LIN {X 0,Y 192.698,Z 291.389,A -85,B 0,C 180,E1 -21893.011,E2 -21893.011} C_VEL
LIN {X 0,Y 200.351,Z 314.138,A -85,B 0,C 180,E1 -21894.699,E2 -21894.699} C_VEL
LIN {X 0,Y 198.491,Z 360.871,A -85,B 0,C 180,E1 -21896.755,E2 -21896.755} C_VEL
LIN {X 0,Y 197.875,Z 372.653,A -85,B 0,C 180,E1 -21897.641,E2 -21897.641} C_VEL
LIN {X 0,Y 196.951,Z 382.953,A -85,B 0,C 180,E1 -21898.798,E2 -21898.798} C_VEL
LIN {X 0,Y 196.113,Z 391.868,A -85,B 0,C 180,E1 -21900.112,E2 -21900.112} C_VEL
LIN {X 0,Y 195.247,Z 399.913,A -85,B 0,C 180,E1 -21901.591,E2 -21901.591} C_VEL
LIN {X 0,Y 194.171,Z 407.148,A -85,B 0,C 180,E1 -21903.2,E2 -21903.2} C_VEL
LIN {X 0,Y 193.185,Z 414.142,A -85,B 0,C 180,E1 -21905.09,E2 -21905.09} C_VEL
LIN {X 0,Y 192.435,Z 419.904,A -85,B 0,C 180,E1 -21906.965,E2 -21906.965} C_VEL
LIN {X 0,Y 191.676,Z 425.271,A -85,B 0,C 180,E1 -21909.054,E2 -21909.054} C_VEL
LIN {X 0,Y 191.095,Z 430.313,A -85,B 0,C 180,E1 -21911.451,E2 -21911.451} C_VEL
LIN {X 0,Y 190.631,Z 434.006,A -85,B 0,C 180,E1 -21913.608,E2 -21913.608} C_VEL
LIN {X 0,Y 190.248,Z 437.996,A -85,B 0,C 180,E1 -21916.63,E2 -21916.63} C_VEL
LIN {X 0,Y 190.193,Z 439.702,A -85,B 0,C 180,E1 -21918.31,E2 -21918.31} C_VEL
LIN {X 0,Y 190.411,Z 441.761,A -85,B 0,C 180,E1 -21921.14,E2 -21921.14} C_VEL
LIN {X 0,Y 190.952,Z 442.925,A -85,B 0,C 180,E1 -21924.065,E2 -21924.065} C_VEL
LIN {X 0,Y 192.023,Z 443.094,A -85,B 0,C 180,E1 -21927.327,E2 -21927.327} C_VEL
LIN {X 0,Y 193.605,Z 442.067,A -85,B 0,C 180,E1 -21930.597,E2 -21930.597} C_VEL
LIN {X 0,Y 196.19,Z 438.937,A -85,B 0,C 180,E1 -21934.543,E2 -21934.543} C_VEL
LIN {X 0,Y 198.352,Z 435.744,A -85,B 0,C 180,E1 -21937.103,E2 -21937.103} C_VEL
LIN {X 0,Y 200.792,Z 431.697,A -85,B 0,C 180,E1 -21939.514,E2 -21939.514} C_VEL
LIN {X 0,Y 204.205,Z 425.453,A -85,B 0,C 180,E1 -21942.311,E2 -21942.311} C_VEL
LIN {X 0,Y 207.631,Z 417.988,A -85,B 0,C 180,E1 -21944.791,E2 -21944.791} C_VEL
LIN {X 0,Y 210.688,Z 410.33,A -85,B 0,C 180,E1 -21946.744,E2 -21946.744} C_VEL
LIN {X 0,Y 212.919,Z 403.856,A -85,B 0,C 180,E1 -21948.096,E2 -21948.096} C_VEL
LIN {X 0,Y 215.546,Z 395.131,A -85,B 0,C 180,E1 -21949.555,E2 -21949.555} C_VEL
LIN {X 0,Y 217.706,Z 386.417,A -85,B 0,C 180,E1 -21950.713,E2 -21950.713} C_VEL
LIN {X 0,Y 219.864,Z 375.243,A -85,B 0,C 180,E1 -21951.841,E2 -21951.841} C_VEL
LIN {X 0,Y 221.31,Z 363.987,A -85,B 0,C 180,E1 -21952.591,E2 -21952.591} C_VEL
LIN {X 0,Y 223.453,Z 336.581,A -85,B 0,C 180,E1 -21953.743,E2 -21953.743} C_VEL
LIN {X 0,Y 217.6,Z 325.466,A -85,B 0,C 180,E1 -21956.298,E2 -21956.298} C_VEL
LIN {X 0,Y 214.117,Z 319.83,A -85,B 0,C 180,E1 -21957.946,E2 -21957.946} C_VEL
LIN {X 0,Y 210.484,Z 314.361,A -85,B 0,C 180,E1 -21959.803,E2 -21959.803} C_VEL
LIN {X 0,Y 208.514,Z 311.193,A -85,B 0,C 180,E1 -21960.926,E2 -21960.926} C_VEL
LIN {X 0,Y 205.81,Z 307.32,A -85,B 0,C 180,E1 -21962.525,E2 -21962.525} C_VEL
LIN {X 0,Y 203.157,Z 304.407,A -85,B 0,C 180,E1 -21964.217,E2 -21964.217} C_VEL
LIN {X 0,Y 202.125,Z 302.631,A -85,B 0,C 180,E1 -21964.988,E2 -21964.988} C_VEL
LIN {X 0,Y 199.456,Z 300.395,A -85,B 0,C 180,E1 -21966.896,E2 -21966.896} C_VEL
LIN {X 0,Y 197.961,Z 297.373,A -85,B 0,C 180,E1 -21968.339,E2 -21968.339} C_VEL
LIN {X 0,Y 194.198,Z 294.632,A -85,B 0,C 180,E1 -21971.987,E2 -21971.987} C_VEL
LIN {X 0,Y 193.008,Z 292.406,A -85,B 0,C 180,E1 -21973.693,E2 -21973.693} C_VEL
LIN {X 0,Y 192.795,Z 291.28,A -85,B 0,C 180,E1 -21974.246,E2 -21974.246} C_VEL
LIN {X 0,Y 192.71,Z 291.289,A -85,B 0,C 180,E1 -21979.163,E2 -21979.163} C_VEL
LIN {X 0,Y 192.662,Z 291.287,A -85,B 0,C 180,E1 -21984.226,E2 -21984.226} C_VEL
LIN {X 0,Y 192.64,Z 291.29,A -85,B 0,C 180,E1 -21988.889,E2 -21988.889} C_VEL
LIN {X 0,Y 193.831,Z 294.774,A -85,B 0,C 180,E1 -21995.462,E2 -21995.462} C_VEL
LIN {X 0,Y 194.221,Z 295.838,A -85,B 0,C 180,E1 -21996.347,E2 -21996.347} C_VEL
LIN {X 0,Y 199.63,Z 303.251,A -85,B 0,C 180,E1 -22001.645,E2 -22001.645} C_VEL
LIN {X 0,Y 203.657,Z 309.45,A -85,B 0,C 180,E1 -22004.662,E2 -22004.662} C_VEL
LIN {X 0,Y 208.105,Z 316.783,A -85,B 0,C 180,E1 -22007.468,E2 -22007.468} C_VEL
LIN {X 0,Y 211.698,Z 323.218,A -85,B 0,C 180,E1 -22009.493,E2 -22009.493} C_VEL
LIN {X 0,Y 215.585,Z 330.908,A -85,B 0,C 180,E1 -22011.482,E2 -22011.482} C_VEL
LIN {X 0,Y 220.085,Z 341.471,A -85,B 0,C 180,E1 -22013.657,E2 -22013.657} C_VEL
LIN {X 0,Y 221.449,Z 354.874,A -85,B 0,C 180,E1 -22014.901,E2 -22014.901} C_VEL
LIN {X 0,Y 221.826,Z 363.402,A -85,B 0,C 180,E1 -22015.531,E2 -22015.531} C_VEL
LIN {X 0,Y 221.197,Z 371.063,A -85,B 0,C 180,E1 -22015.822,E2 -22015.822} C_VEL
LIN {X 0,Y 220.14,Z 376.884,A -85,B 0,C 180,E1 -22015.915,E2 -22015.915} C_VEL
LIN {X 0,Y 216.946,Z 386.292,A -85,B 0,C 180,E1 -22015.875,E2 -22015.875} C_VEL
LIN {X 0,Y 213.279,Z 395.447,A -85,B 0,C 180,E1 -22016.008,E2 -22016.008} C_VEL
LIN {X 0,Y 211.5,Z 400.855,A -85,B 0,C 180,E1 -22016.403,E2 -22016.403} C_VEL
LIN {X 0,Y 208.494,Z 411.167,A -85,B 0,C 180,E1 -22017.649,E2 -22017.649} C_VEL
LIN {X 0,Y 205.745,Z 419.123,A -85,B 0,C 180,E1 -22018.893,E2 -22018.893} C_VEL
LIN {X 0,Y 202.813,Z 426.763,A -85,B 0,C 180,E1 -22020.411,E2 -22020.411} C_VEL
LIN {X 0,Y 198.982,Z 435.728,A -85,B 0,C 180,E1 -22022.668,E2 -22022.668} C_VEL
LIN {X 0,Y 195.446,Z 442.776,A -85,B 0,C 180,E1 -22025.008,E2 -22025.008} C_VEL
LIN {X 0,Y 192.345,Z 448.444,A -85,B 0,C 180,E1 -22027.441,E2 -22027.441} C_VEL
LIN {X 0,Y 189.195,Z 453.782,A -85,B 0,C 180,E1 -22030.47,E2 -22030.47} C_VEL
LIN {X 0,Y 186.736,Z 457.778,A -85,B 0,C 180,E1 -22033.605,E2 -22033.605} C_VEL
LIN {X 0,Y 184.977,Z 460.546,A -85,B 0,C 180,E1 -22036.824,E2 -22036.824} C_VEL
LIN {X 0,Y 184.163,Z 461.689,A -85,B 0,C 180,E1 -22039.001,E2 -22039.001} C_VEL
LIN {X 0,Y 183.645,Z 462.356,A -85,B 0,C 180,E1 -22041.195,E2 -22041.195} C_VEL
LIN {X 0,Y 183.328,Z 462.409,A -85,B 0,C 180,E1 -22045.381,E2 -22045.381} C_VEL
LIN {X 0,Y 183.47,Z 461.54,A -85,B 0,C 180,E1 -22047.805,E2 -22047.805} C_VEL
LIN {X 0,Y 183.571,Z 460.179,A -85,B 0,C 180,E1 -22050.001,E2 -22050.001} C_VEL
LIN {X 0,Y 183.601,Z 457.145,A -85,B 0,C 180,E1 -22053.292,E2 -22053.292} C_VEL
LIN {X 0,Y 183.609,Z 452.606,A -85,B 0,C 180,E1 -22056.594,E2 -22056.594} C_VEL
LIN {X 0,Y 183.92,Z 447.511,A -85,B 0,C 180,E1 -22059.347,E2 -22059.347} C_VEL
LIN {X 0,Y 184.381,Z 442.506,A -85,B 0,C 180,E1 -22061.544,E2 -22061.544} C_VEL
LIN {X 0,Y 185.122,Z 436.463,A -85,B 0,C 180,E1 -22063.726,E2 -22063.726} C_VEL
LIN {X 0,Y 186.263,Z 428.077,A -85,B 0,C 180,E1 -22066.157,E2 -22066.157} C_VEL
LIN {X 0,Y 187.402,Z 420.033,A -85,B 0,C 180,E1 -22068.023,E2 -22068.023} C_VEL
LIN {X 0,Y 188.624,Z 409.933,A -85,B 0,C 180,E1 -22069.876,E2 -22069.876} C_VEL
LIN {X 0,Y 189.99,Z 399.38,A -85,B 0,C 180,E1 -22071.283,E2 -22071.283} C_VEL
LIN {X 0,Y 190.803,Z 389.702,A -85,B 0,C 180,E1 -22072.245,E2 -22072.245} C_VEL
LIN {X 0,Y 191.446,Z 379.539,A -85,B 0,C 180,E1 -22072.939,E2 -22072.939} C_VEL
LIN {X 0,Y 192.199,Z 354.528,A -85,B 0,C 180,E1 -22074.102,E2 -22074.102} C_VEL
LIN {X 0,Y 187.917,Z 303.799,A -85,B 0,C 180,E1 -22076.892,E2 -22076.892} C_VEL
LIN {X 0,Y 186.171,Z 294.826,A -85,B 0,C 180,E1 -22081.396,E2 -22081.396} C_VEL
LIN {X 0,Y 185.691,Z 292.169,A -85,B 0,C 180,E1 -22082.815,E2 -22082.815} C_VEL
LIN {X 0,Y 185.548,Z 292.184,A -85,B 0,C 180,E1 -22087.303,E2 -22087.303} C_VEL
LIN {X 0,Y 185.488,Z 292.19,A -85,B 0,C 180,E1 -22090.729,E2 -22090.729} C_VEL
LIN {X 0,Y 185.462,Z 292.195,A -85,B 0,C 180,E1 -22096.054,E2 -22096.054} C_VEL
LIN {X 0,Y 185.469,Z 292.192,A -85,B 0,C 180,E1 -22099.894,E2 -22099.894} C_VEL
LIN {X 0,Y 185.508,Z 292.186,A -85,B 0,C 180,E1 -22102.71,E2 -22102.71} C_VEL
LIN {X 0,Y 185.545,Z 292.183,A -85,B 0,C 180,E1 -22107.973,E2 -22107.973} C_VEL
LIN {X 0,Y 185.583,Z 292.175,A -85,B 0,C 180,E1 -22110.575,E2 -22110.575} C_VEL
LIN {X 0,Y 185.589,Z 292.18,A -85,B 0,C 180,E1 -22115.381,E2 -22115.381} C_VEL
LIN {X 0,Y 185.675,Z 292.167,A -85,B 0,C 180,E1 -22121.132,E2 -22121.132} C_VEL
LIN {X 0,Y 185.694,Z 292.164,A -85,B 0,C 180,E1 -22124.635,E2 -22124.635} C_VEL
LIN {X 0,Y 185.888,Z 292.141,A -85,B 0,C 180,E1 -22129.416,E2 -22129.416} C_VEL
LIN {X 0,Y 185.947,Z 292.135,A -85,B 0,C 180,E1 -22133.488,E2 -22133.488} C_VEL
LIN {X 0,Y 186.205,Z 292.103,A -85,B 0,C 180,E1 -22137.835,E2 -22137.835} C_VEL
LIN {X 0,Y 186.405,Z 292.078,A -85,B 0,C 180,E1 -22139.998,E2 -22139.998} C_VEL
LIN {X 0,Y 185.923,Z 292.134,A -85,B 0,C 180,E1 -22144.334,E2 -22144.334} C_VEL
LIN {X 0,Y 186.011,Z 292.125,A -85,B 0,C 180,E1 -22148.691,E2 -22148.691} C_VEL
LIN {X 0,Y 185.731,Z 292.157,A -85,B 0,C 180,E1 -22153.121,E2 -22153.121} C_VEL
LIN {X 0,Y 185.707,Z 292.162,A -85,B 0,C 180,E1 -22158.897,E2 -22158.897} C_VEL
LIN {X 0,Y 185.597,Z 292.177,A -85,B 0,C 180,E1 -22164.66,E2 -22164.66} C_VEL
LIN {X 0,Y 185.575,Z 292.178,A -85,B 0,C 180,E1 -22169.491,E2 -22169.491} C_VEL
LIN {X 0,Y 185.516,Z 292.187,A -85,B 0,C 180,E1 -22174.626,E2 -22174.626} C_VEL
LIN {X 0,Y 185.539,Z 292.183,A -85,B 0,C 180,E1 -22177.302,E2 -22177.302} C_VEL
LIN {X 0,Y 185.524,Z 292.186,A -85,B 0,C 180,E1 -22180.744,E2 -22180.744} C_VEL
LIN {X 0,Y 185.559,Z 292.179,A -85,B 0,C 180,E1 -22186.02,E2 -22186.02} C_VEL
LIN {X 0,Y 185.536,Z 292.187,A -85,B 0,C 180,E1 -22189.913,E2 -22189.913} C_VEL
LIN {X 0,Y 185.554,Z 292.181,A -85,B 0,C 180,E1 -22192.699,E2 -22192.699} C_VEL
LIN {X 0,Y 185.539,Z 292.186,A -85,B 0,C 180,E1 -22197.974,E2 -22197.974} C_VEL
LIN {X 0,Y 185.576,Z 292.179,A -85,B 0,C 180,E1 -22200.575,E2 -22200.575} C_VEL
LIN {X 0,Y 185.581,Z 292.178,A -85,B 0,C 180,E1 -22205.382,E2 -22205.382} C_VEL
LIN {X 0,Y 185.669,Z 292.166,A -85,B 0,C 180,E1 -22211.132,E2 -22211.132} C_VEL
LIN {X 0,Y 185.718,Z 292.162,A -85,B 0,C 180,E1 -22214.639,E2 -22214.639} C_VEL
LIN {X 0,Y 185.918,Z 292.136,A -85,B 0,C 180,E1 -22219.358,E2 -22219.358} C_VEL
LIN {X 0,Y 185.954,Z 292.134,A -85,B 0,C 180,E1 -22223.489,E2 -22223.489} C_VEL
LIN {X 0,Y 186.2,Z 292.1,A -85,B 0,C 180,E1 -22227.836,E2 -22227.836} C_VEL
LIN {X 0,Y 186.4,Z 292.077,A -85,B 0,C 180,E1 -22229.999,E2 -22229.999} C_VEL
LIN {X 0,Y 185.916,Z 292.137,A -85,B 0,C 180,E1 -22234.335,E2 -22234.335} C_VEL
LIN {X 0,Y 186.001,Z 292.125,A -85,B 0,C 180,E1 -22238.692,E2 -22238.692} C_VEL
LIN {X 0,Y 185.757,Z 292.157,A -85,B 0,C 180,E1 -22243.12,E2 -22243.12} C_VEL
LIN {X 0,Y 185.682,Z 292.169,A -85,B 0,C 180,E1 -22247.625,E2 -22247.625} C_VEL
LIN {X 0,Y 185.609,Z 292.177,A -85,B 0,C 180,E1 -22252.395,E2 -22252.395} C_VEL
LIN {X 0,Y 193.402,Z 315.234,A -85,B 0,C 180,E1 -22254.206,E2 -22254.206} C_VEL
LIN {X 0,Y 191.595,Z 360.842,A -85,B 0,C 180,E1 -22256.287,E2 -22256.287} C_VEL
LIN {X 0,Y 190.952,Z 372.604,A -85,B 0,C 180,E1 -22257.185,E2 -22257.185} C_VEL
LIN {X 0,Y 189.931,Z 383.741,A -85,B 0,C 180,E1 -22258.481,E2 -22258.481} C_VEL
LIN {X 0,Y 189.094,Z 392.381,A -85,B 0,C 180,E1 -22259.807,E2 -22259.807} C_VEL
LIN {X 0,Y 188.286,Z 399.565,A -85,B 0,C 180,E1 -22261.159,E2 -22261.159} C_VEL
LIN {X 0,Y 187.086,Z 407.606,A -85,B 0,C 180,E1 -22263.003,E2 -22263.003} C_VEL
LIN {X 0,Y 186.151,Z 414.112,A -85,B 0,C 180,E1 -22264.821,E2 -22264.821} C_VEL
LIN {X 0,Y 185.456,Z 419.331,A -85,B 0,C 180,E1 -22266.543,E2 -22266.543} C_VEL
LIN {X 0,Y 184.608,Z 425.155,A -85,B 0,C 180,E1 -22268.847,E2 -22268.847} C_VEL
LIN {X 0,Y 184.064,Z 429.983,A -85,B 0,C 180,E1 -22271.172,E2 -22271.172} C_VEL
LIN {X 0,Y 183.527,Z 434.046,A -85,B 0,C 180,E1 -22273.572,E2 -22273.572} C_VEL
LIN {X 0,Y 183.192,Z 437.698,A -85,B 0,C 180,E1 -22276.329,E2 -22276.329} C_VEL
LIN {X 0,Y 183.143,Z 440.57,A -85,B 0,C 180,E1 -22279.283,E2 -22279.283} C_VEL
LIN {X 0,Y 183.707,Z 443.063,A -85,B 0,C 180,E1 -22283.453,E2 -22283.453} C_VEL
LIN {X 0,Y 184.706,Z 443.638,A -85,B 0,C 180,E1 -22286.831,E2 -22286.831} C_VEL
LIN {X 0,Y 186.495,Z 442.813,A -85,B 0,C 180,E1 -22290.668,E2 -22290.668} C_VEL
LIN {X 0,Y 189.185,Z 440.155,A -85,B 0,C 180,E1 -22294.81,E2 -22294.81} C_VEL
LIN {X 0,Y 191.728,Z 436.783,A -85,B 0,C 180,E1 -22297.764,E2 -22297.764} C_VEL
LIN {X 0,Y 194.21,Z 432.995,A -85,B 0,C 180,E1 -22300.195,E2 -22300.195} C_VEL
LIN {X 0,Y 196.798,Z 428.706,A -85,B 0,C 180,E1 -22302.323,E2 -22302.323} C_VEL
LIN {X 0,Y 200.044,Z 422.512,A -85,B 0,C 180,E1 -22304.725,E2 -22304.725} C_VEL
LIN {X 0,Y 202.863,Z 416.534,A -85,B 0,C 180,E1 -22306.569,E2 -22306.569} C_VEL
LIN {X 0,Y 206.102,Z 408.688,A -85,B 0,C 180,E1 -22308.51,E2 -22308.51} C_VEL
LIN {X 0,Y 209.448,Z 399.12,A -85,B 0,C 180,E1 -22310.343,E2 -22310.343} C_VEL
LIN {X 0,Y 212.119,Z 389.409,A -85,B 0,C 180,E1 -22311.746,E2 -22311.746} C_VEL
LIN {X 0,Y 214.281,Z 379.683,A -85,B 0,C 180,E1 -22312.809,E2 -22312.809} C_VEL
LIN {X 0,Y 215.719,Z 370.797,A -85,B 0,C 180,E1 -22313.557,E2 -22313.557} C_VEL
LIN {X 0,Y 217.003,Z 359.592,A -85,B 0,C 180,E1 -22314.202,E2 -22314.202} C_VEL
LIN {X 0,Y 218.549,Z 339.503,A -85,B 0,C 180,E1 -22315.032,E2 -22315.032} C_VEL
LIN {X 0,Y 213.644,Z 329.87,A -85,B 0,C 180,E1 -22317.38,E2 -22317.38} C_VEL
LIN {X 0,Y 210.475,Z 324.818,A -85,B 0,C 180,E1 -22318.96,E2 -22318.96} C_VEL
LIN {X 0,Y 205.715,Z 317.082,A -85,B 0,C 180,E1 -22321.704,E2 -22321.704} C_VEL
LIN {X 0,Y 203.329,Z 313.604,A -85,B 0,C 180,E1 -22323.211,E2 -22323.211} C_VEL
LIN {X 0,Y 200.543,Z 310.193,A -85,B 0,C 180,E1 -22325.122,E2 -22325.122} C_VEL
LIN {X 0,Y 199.619,Z 308.946,A -85,B 0,C 180,E1 -22325.811,E2 -22325.811} C_VEL
LIN {X 0,Y 196.979,Z 306.174,A -85,B 0,C 180,E1 -22327.932,E2 -22327.932} C_VEL
LIN {X 0,Y 195.858,Z 303.828,A -85,B 0,C 180,E1 -22329.095,E2 -22329.095} C_VEL
LIN {X 0,Y 192.674,Z 301.456,A -85,B 0,C 180,E1 -22332.365,E2 -22332.365} C_VEL
LIN {X 0,Y 191.317,Z 298.86,A -85,B 0,C 180,E1 -22334.426,E2 -22334.426} C_VEL
LIN {X 0,Y 191.071,Z 298.182,A -85,B 0,C 180,E1 -22334.922,E2 -22334.922} C_VEL
LIN {X 0,Y 188.225,Z 296.835,A -85,B 0,C 180,E1 -22341.926,E2 -22341.926} C_VEL
LIN {X 0,Y 188.284,Z 296.943,A -85,B 0,C 180,E1 -22346.612,E2 -22346.612} C_VEL
LIN {X 0,Y 188.963,Z 297.537,A -85,B 0,C 180,E1 -22349.221,E2 -22349.221} C_VEL
LIN {X 0,Y 192.232,Z 301.815,A -85,B 0,C 180,E1 -22355.319,E2 -22355.319} C_VEL
LIN {X 0,Y 197.076,Z 308.988,A -85,B 0,C 180,E1 -22360.605,E2 -22360.605} C_VEL
LIN {X 0,Y 201.683,Z 316.494,A -85,B 0,C 180,E1 -22364.286,E2 -22364.286} C_VEL
LIN {X 0,Y 205.401,Z 322.922,A -85,B 0,C 180,E1 -22366.76,E2 -22366.76} C_VEL
LIN {X 0,Y 208.337,Z 328.367,A -85,B 0,C 180,E1 -22368.53,E2 -22368.53} C_VEL
LIN {X 0,Y 212.02,Z 336.084,A -85,B 0,C 180,E1 -22370.57,E2 -22370.57} C_VEL
LIN {X 0,Y 215.656,Z 345.058,A -85,B 0,C 180,E1 -22372.499,E2 -22372.499} C_VEL
LIN {X 0,Y 216.746,Z 357.398,A -85,B 0,C 180,E1 -22373.663,E2 -22373.663} C_VEL
LIN {X 0,Y 216.993,Z 364.53,A -85,B 0,C 180,E1 -22374.197,E2 -22374.197} C_VEL
LIN {X 0,Y 215.208,Z 382.567,A -85,B 0,C 180,E1 -22374.972,E2 -22374.972} C_VEL
LIN {X 0,Y 213.235,Z 393.234,A -85,B 0,C 180,E1 -22375.697,E2 -22375.697} C_VEL
LIN {X 0,Y 211.5,Z 400.855,A -85,B 0,C 180,E1 -22376.403,E2 -22376.403} C_VEL
LIN {X 0,Y 209.976,Z 404.484,A -85,B 0,C 180,E1 -22376.651,E2 -22376.651} C_VEL
LIN {X 0,Y 206.162,Z 410.158,A -85,B 0,C 180,E1 -22376.796,E2 -22376.796} C_VEL
LIN {X 0,Y 202.253,Z 415.631,A -85,B 0,C 180,E1 -22377.027,E2 -22377.027} C_VEL
LIN {X 0,Y 200.604,Z 418.76,A -85,B 0,C 180,E1 -22377.456,E2 -22377.456} C_VEL
LIN {X 0,Y 197.188,Z 427.239,A -85,B 0,C 180,E1 -22379.181,E2 -22379.181} C_VEL
LIN {X 0,Y 192.766,Z 436.673,A -85,B 0,C 180,E1 -22381.709,E2 -22381.709} C_VEL
LIN {X 0,Y 189.083,Z 443.41,A -85,B 0,C 180,E1 -22384.105,E2 -22384.105} C_VEL
LIN {X 0,Y 185.84,Z 448.869,A -85,B 0,C 180,E1 -22386.605,E2 -22386.605} C_VEL
LIN {X 0,Y 183.563,Z 452.459,A -85,B 0,C 180,E1 -22388.672,E2 -22388.672} C_VEL
LIN {X 0,Y 180.691,Z 456.661,A -85,B 0,C 180,E1 -22391.872,E2 -22391.872} C_VEL
LIN {X 0,Y 179.219,Z 458.757,A -85,B 0,C 180,E1 -22394.069,E2 -22394.069} C_VEL
LIN {X 0,Y 178.055,Z 460.375,A -85,B 0,C 180,E1 -22396.302,E2 -22396.302} C_VEL
LIN {X 0,Y 177.189,Z 461.48,A -85,B 0,C 180,E1 -22398.562,E2 -22398.562} C_VEL
LIN {X 0,Y 176.613,Z 462.017,A -85,B 0,C 180,E1 -22400.842,E2 -22400.842} C_VEL
LIN {X 0,Y 176.31,Z 462.112,A -85,B 0,C 180,E1 -22403.133,E2 -22403.133} C_VEL
LIN {X 0,Y 176.265,Z 461.764,A -85,B 0,C 180,E1 -22405.427,E2 -22405.427} C_VEL
LIN {X 0,Y 176.403,Z 460.922,A -85,B 0,C 180,E1 -22407.717,E2 -22407.717} C_VEL
LIN {X 0,Y 176.48,Z 458.525,A -85,B 0,C 180,E1 -22411.141,E2 -22411.141} C_VEL
LIN {X 0,Y 176.544,Z 456.246,A -85,B 0,C 180,E1 -22413.424,E2 -22413.424} C_VEL
LIN {X 0,Y 176.587,Z 451.438,A -85,B 0,C 180,E1 -22416.858,E2 -22416.858} C_VEL
LIN {X 0,Y 176.926,Z 446.182,A -85,B 0,C 180,E1 -22419.72,E2 -22419.72} C_VEL
LIN {X 0,Y 177.435,Z 440.999,A -85,B 0,C 180,E1 -22422.002,E2 -22422.002} C_VEL
LIN {X 0,Y 178.222,Z 434.749,A -85,B 0,C 180,E1 -22424.268,E2 -22424.268} C_VEL
LIN {X 0,Y 179.301,Z 427.158,A -85,B 0,C 180,E1 -22426.51,E2 -22426.51} C_VEL
LIN {X 0,Y 180.671,Z 417.781,A -85,B 0,C 180,E1 -22428.719,E2 -22428.719} C_VEL
LIN {X 0,Y 181.754,Z 408.679,A -85,B 0,C 180,E1 -22430.366,E2 -22430.366} C_VEL
LIN {X 0,Y 183.03,Z 399.064,A -85,B 0,C 180,E1 -22431.69,E2 -22431.69} C_VEL
LIN {X 0,Y 183.892,Z 389.191,A -85,B 0,C 180,E1 -22432.706,E2 -22432.706} C_VEL
LIN {X 0,Y 184.511,Z 379.499,A -85,B 0,C 180,E1 -22433.395,E2 -22433.395} C_VEL
LIN {X 0,Y 185.33,Z 355.521,A -85,B 0,C 180,E1 -22434.555,E2 -22434.555} C_VEL
LIN {X 0,Y 181.15,Z 305.379,A -85,B 0,C 180,E1 -22437.414,E2 -22437.414} C_VEL
LIN {X 0,Y 180.607,Z 303.059,A -85,B 0,C 180,E1 -22437.623,E2 -22437.623} C_VEL
LIN {X 0,Y 178.625,Z 293.049,A -85,B 0,C 180,E1 -22443.087,E2 -22443.087} C_VEL
LIN {X 0,Y 178.422,Z 293.072,A -85,B 0,C 180,E1 -22449.067,E2 -22449.067} C_VEL
LIN {X 0,Y 178.406,Z 293.07,A -85,B 0,C 180,E1 -22452.042,E2 -22452.042} C_VEL
LIN {X 0,Y 178.396,Z 293.073,A -85,B 0,C 180,E1 -22455.163,E2 -22455.163} C_VEL
LIN {X 0,Y 178.405,Z 293.073,A -85,B 0,C 180,E1 -22458.458,E2 -22458.458} C_VEL
LIN {X 0,Y 178.424,Z 293.073,A -85,B 0,C 180,E1 -22463.781,E2 -22463.781} C_VEL
LIN {X 0,Y 178.487,Z 293.063,A -85,B 0,C 180,E1 -22466.545,E2 -22466.545} C_VEL
LIN {X 0,Y 178.524,Z 293.056,A -85,B 0,C 180,E1 -22470.005,E2 -22470.005} C_VEL
LIN {X 0,Y 178.536,Z 293.057,A -85,B 0,C 180,E1 -22474.874,E2 -22474.874} C_VEL
LIN {X 0,Y 178.624,Z 293.045,A -85,B 0,C 180,E1 -22480.782,E2 -22480.782} C_VEL
LIN {X 0,Y 178.657,Z 293.037,A -85,B 0,C 180,E1 -22486.346,E2 -22486.346} C_VEL
LIN {X 0,Y 178.911,Z 293.01,A -85,B 0,C 180,E1 -22490.958,E2 -22490.958} C_VEL
LIN {X 0,Y 179.151,Z 292.982,A -85,B 0,C 180,E1 -22497.75,E2 -22497.75} C_VEL
LIN {X 0,Y 179.368,Z 292.954,A -85,B 0,C 180,E1 -22499.998,E2 -22499.998} C_VEL
LIN {X 0,Y 178.871,Z 293.012,A -85,B 0,C 180,E1 -22504.505,E2 -22504.505} C_VEL
LIN {X 0,Y 178.961,Z 293.004,A -85,B 0,C 180,E1 -22509.036,E2 -22509.036} C_VEL
LIN {X 0,Y 178.659,Z 293.04,A -85,B 0,C 180,E1 -22513.65,E2 -22513.65} C_VEL
LIN {X 0,Y 178.65,Z 293.042,A -85,B 0,C 180,E1 -22519.242,E2 -22519.242} C_VEL
LIN {X 0,Y 178.531,Z 293.058,A -85,B 0,C 180,E1 -22525.123,E2 -22525.123} C_VEL
LIN {X 0,Y 178.475,Z 293.062,A -85,B 0,C 180,E1 -22530.789,E2 -22530.789} C_VEL
LIN {X 0,Y 178.492,Z 293.063,A -85,B 0,C 180,E1 -22534.223,E2 -22534.223} C_VEL
LIN {X 0,Y 178.439,Z 293.066,A -85,B 0,C 180,E1 -22539.06,E2 -22539.06} C_VEL
LIN {X 0,Y 178.482,Z 293.065,A -85,B 0,C 180,E1 -22542.018,E2 -22542.018} C_VEL
LIN {X 0,Y 178.512,Z 293.058,A -85,B 0,C 180,E1 -22545.123,E2 -22545.123} C_VEL
LIN {X 0,Y 178.497,Z 293.061,A -85,B 0,C 180,E1 -22548.422,E2 -22548.422} C_VEL
LIN {X 0,Y 178.453,Z 293.065,A -85,B 0,C 180,E1 -22553.79,E2 -22553.79} C_VEL
LIN {X 0,Y 178.486,Z 293.062,A -85,B 0,C 180,E1 -22556.547,E2 -22556.547} C_VEL
LIN {X 0,Y 178.517,Z 293.06,A -85,B 0,C 180,E1 -22560.005,E2 -22560.005} C_VEL
LIN {X 0,Y 178.529,Z 293.056,A -85,B 0,C 180,E1 -22564.875,E2 -22564.875} C_VEL
LIN {X 0,Y 178.617,Z 293.044,A -85,B 0,C 180,E1 -22570.783,E2 -22570.783} C_VEL
LIN {X 0,Y 178.659,Z 293.043,A -85,B 0,C 180,E1 -22574.016,E2 -22574.016} C_VEL
LIN {X 0,Y 178.855,Z 293.015,A -85,B 0,C 180,E1 -22579.209,E2 -22579.209} C_VEL
LIN {X 0,Y 178.918,Z 293.009,A -85,B 0,C 180,E1 -22583.232,E2 -22583.232} C_VEL
LIN {X 0,Y 179.146,Z 292.979,A -85,B 0,C 180,E1 -22587.751,E2 -22587.751} C_VEL
LIN {X 0,Y 179.363,Z 292.954,A -85,B 0,C 180,E1 -22589.999,E2 -22589.999} C_VEL
LIN {X 0,Y 178.864,Z 293.015,A -85,B 0,C 180,E1 -22594.507,E2 -22594.507} C_VEL
LIN {X 0,Y 178.952,Z 293.003,A -85,B 0,C 180,E1 -22599.037,E2 -22599.037} C_VEL
LIN {X 0,Y 178.68,Z 293.04,A -85,B 0,C 180,E1 -22603.65,E2 -22603.65} C_VEL
LIN {X 0,Y 178.635,Z 293.044,A -85,B 0,C 180,E1 -22608.344,E2 -22608.344} C_VEL
LIN {X 0,Y 178.549,Z 293.057,A -85,B 0,C 180,E1 -22611.806,E2 -22611.806} C_VEL
LIN {X 0,Y 186.632,Z 316.9,A -85,B 0,C 180,E1 -22613.73,E2 -22613.73} C_VEL
LIN {X 0,Y 184.655,Z 361.399,A -85,B 0,C 180,E1 -22615.841,E2 -22615.841} C_VEL
LIN {X 0,Y 184.076,Z 371.745,A -85,B 0,C 180,E1 -22616.653,E2 -22616.653} C_VEL
LIN {X 0,Y 182.96,Z 384.023,A -85,B 0,C 180,E1 -22618.098,E2 -22618.098} C_VEL
LIN {X 0,Y 182.011,Z 393.352,A -85,B 0,C 180,E1 -22619.598,E2 -22619.598} C_VEL
LIN {X 0,Y 180.947,Z 401.791,A -85,B 0,C 180,E1 -22621.302,E2 -22621.302} C_VEL
LIN {X 0,Y 179.598,Z 410.629,A -85,B 0,C 180,E1 -22623.516,E2 -22623.516} C_VEL
LIN {X 0,Y 178.438,Z 418.999,A -85,B 0,C 180,E1 -22626.212,E2 -22626.212} C_VEL
LIN {X 0,Y 177.612,Z 424.689,A -85,B 0,C 180,E1 -22628.484,E2 -22628.484} C_VEL
LIN {X 0,Y 176.999,Z 429.902,A -85,B 0,C 180,E1 -22631.029,E2 -22631.029} C_VEL
LIN {X 0,Y 176.333,Z 434.957,A -85,B 0,C 180,E1 -22634.162,E2 -22634.162} C_VEL
LIN {X 0,Y 176.024,Z 438.74,A -85,B 0,C 180,E1 -22637.257,E2 -22637.257} C_VEL
LIN {X 0,Y 176.119,Z 441.438,A -85,B 0,C 180,E1 -22640.325,E2 -22640.325} C_VEL
LIN {X 0,Y 176.575,Z 443.148,A -85,B 0,C 180,E1 -22643.346,E2 -22643.346} C_VEL
LIN {X 0,Y 177.404,Z 443.964,A -85,B 0,C 180,E1 -22646.318,E2 -22646.318} C_VEL
LIN {X 0,Y 178.853,Z 443.87,A -85,B 0,C 180,E1 -22649.821,E2 -22649.821} C_VEL
LIN {X 0,Y 180.915,Z 442.453,A -85,B 0,C 180,E1 -22653.31,E2 -22653.31} C_VEL
LIN {X 0,Y 183.548,Z 439.68,A -85,B 0,C 180,E1 -22656.769,E2 -22656.769} C_VEL
LIN {X 0,Y 186.852,Z 435.408,A -85,B 0,C 180,E1 -22660.216,E2 -22660.216} C_VEL
LIN {X 0,Y 190.704,Z 429.671,A -85,B 0,C 180,E1 -22663.365,E2 -22663.365} C_VEL
LIN {X 0,Y 194.391,Z 423.134,A -85,B 0,C 180,E1 -22665.995,E2 -22665.995} C_VEL
LIN {X 0,Y 197.03,Z 417.963,A -85,B 0,C 180,E1 -22667.644,E2 -22667.644} C_VEL
LIN {X 0,Y 200.148,Z 410.948,A -85,B 0,C 180,E1 -22669.471,E2 -22669.471} C_VEL
LIN {X 0,Y 202.993,Z 403.495,A -85,B 0,C 180,E1 -22671.039,E2 -22671.039} C_VEL
LIN {X 0,Y 206.209,Z 393.646,A -85,B 0,C 180,E1 -22672.659,E2 -22672.659} C_VEL
LIN {X 0,Y 208.993,Z 382.773,A -85,B 0,C 180,E1 -22673.97,E2 -22673.97} C_VEL
LIN {X 0,Y 210.766,Z 373.08,A -85,B 0,C 180,E1 -22674.857,E2 -22674.857} C_VEL
LIN {X 0,Y 212.092,Z 363.276,A -85,B 0,C 180,E1 -22675.474,E2 -22675.474} C_VEL
LIN {X 0,Y 213.947,Z 342.669,A -85,B 0,C 180,E1 -22676.351,E2 -22676.351} C_VEL
LIN {X 0,Y 209.183,Z 333.308,A -85,B 0,C 180,E1 -22678.809,E2 -22678.809} C_VEL
LIN {X 0,Y 202.947,Z 323.019,A -85,B 0,C 180,E1 -22682.497,E2 -22682.497} C_VEL
LIN {X 0,Y 200.754,Z 319.7,A -85,B 0,C 180,E1 -22684.017,E2 -22684.017} C_VEL
LIN {X 0,Y 198.045,Z 316.092,A -85,B 0,C 180,E1 -22685.998,E2 -22685.998} C_VEL
LIN {X 0,Y 194.748,Z 312.196,A -85,B 0,C 180,E1 -22688.83,E2 -22688.83} C_VEL
LIN {X 0,Y 193.81,Z 310.422,A -85,B 0,C 180,E1 -22689.83,E2 -22689.83} C_VEL
LIN {X 0,Y 190.859,Z 307.86,A -85,B 0,C 180,E1 -22693.172,E2 -22693.172} C_VEL
LIN {X 0,Y 189.557,Z 305.072,A -85,B 0,C 180,E1 -22695.433,E2 -22695.433} C_VEL
LIN {X 0,Y 187.058,Z 303.807,A -85,B 0,C 180,E1 -22702.07,E2 -22702.07} C_VEL
LIN {X 0,Y 187.168,Z 303.955,A -85,B 0,C 180,E1 -22706.783,E2 -22706.783} C_VEL
LIN {X 0,Y 187.755,Z 304.576,A -85,B 0,C 180,E1 -22709.12,E2 -22709.12} C_VEL
LIN {X 0,Y 190.665,Z 308.622,A -85,B 0,C 180,E1 -22714.845,E2 -22714.845} C_VEL
LIN {X 0,Y 195.398,Z 316.095,A -85,B 0,C 180,E1 -22720.283,E2 -22720.283} C_VEL
LIN {X 0,Y 199.261,Z 322.715,A -85,B 0,C 180,E1 -22723.544,E2 -22723.544} C_VEL
LIN {X 0,Y 202.506,Z 328.64,A -85,B 0,C 180,E1 -22725.886,E2 -22725.886} C_VEL
LIN {X 0,Y 205.513,Z 334.477,A -85,B 0,C 180,E1 -22727.807,E2 -22727.807} C_VEL
LIN {X 0,Y 209.544,Z 343.651,A -85,B 0,C 180,E1 -22730.206,E2 -22730.206} C_VEL
LIN {X 0,Y 211.472,Z 348.859,A -85,B 0,C 180,E1 -22731.304,E2 -22731.304} C_VEL
LIN {X 0,Y 212.37,Z 363.132,A -85,B 0,C 180,E1 -22732.639,E2 -22732.639} C_VEL
LIN {X 0,Y 211.883,Z 370.305,A -85,B 0,C 180,E1 -22732.975,E2 -22732.975} C_VEL
LIN {X 0,Y 210.116,Z 384.489,A -85,B 0,C 180,E1 -22733.663,E2 -22733.663} C_VEL
LIN {X 0,Y 208.198,Z 394.072,A -85,B 0,C 180,E1 -22734.354,E2 -22734.354} C_VEL
LIN {X 0,Y 206.132,Z 402.404,A -85,B 0,C 180,E1 -22735.176,E2 -22735.176} C_VEL
LIN {X 0,Y 203.583,Z 410.576,A -85,B 0,C 180,E1 -22736.176,E2 -22736.176} C_VEL
LIN {X 0,Y 200.604,Z 418.76,A -85,B 0,C 180,E1 -22737.456,E2 -22737.456} C_VEL
LIN {X 0,Y 198.345,Z 423.523,A -85,B 0,C 180,E1 -22738.252,E2 -22738.252} C_VEL
LIN {X 0,Y 192.936,Z 430.835,A -85,B 0,C 180,E1 -22739.389,E2 -22739.389} C_VEL
LIN {X 0,Y 187.239,Z 437.529,A -85,B 0,C 180,E1 -22740.762,E2 -22740.762} C_VEL
LIN {X 0,Y 184.583,Z 441.18,A -85,B 0,C 180,E1 -22741.929,E2 -22741.929} C_VEL
LIN {X 0,Y 180.697,Z 447.405,A -85,B 0,C 180,E1 -22744.671,E2 -22744.671} C_VEL
LIN {X 0,Y 176.968,Z 452.753,A -85,B 0,C 180,E1 -22747.836,E2 -22747.836} C_VEL
LIN {X 0,Y 173.957,Z 456.766,A -85,B 0,C 180,E1 -22751.144,E2 -22751.144} C_VEL
LIN {X 0,Y 172.379,Z 458.711,A -85,B 0,C 180,E1 -22753.419,E2 -22753.419} C_VEL
LIN {X 0,Y 171.156,Z 460.181,A -85,B 0,C 180,E1 -22755.738,E2 -22755.738} C_VEL
LIN {X 0,Y 170.206,Z 461.205,A -85,B 0,C 180,E1 -22758.086,E2 -22758.086} C_VEL
LIN {X 0,Y 169.603,Z 461.685,A -85,B 0,C 180,E1 -22760.46,E2 -22760.46} C_VEL
LIN {X 0,Y 169.251,Z 461.636,A -85,B 0,C 180,E1 -22762.845,E2 -22762.845} C_VEL
LIN {X 0,Y 169.224,Z 461.108,A -85,B 0,C 180,E1 -22765.39,E2 -22765.39} C_VEL
LIN {X 0,Y 169.337,Z 460.225,A -85,B 0,C 180,E1 -22767.622,E2 -22767.622} C_VEL
LIN {X 0,Y 169.442,Z 458.713,A -85,B 0,C 180,E1 -22770.001,E2 -22770.001} C_VEL
LIN {X 0,Y 169.488,Z 455.255,A -85,B 0,C 180,E1 -22773.567,E2 -22773.567} C_VEL
LIN {X 0,Y 169.511,Z 451.487,A -85,B 0,C 180,E1 -22776.382,E2 -22776.382} C_VEL
LIN {X 0,Y 169.81,Z 446.004,A -85,B 0,C 180,E1 -22779.53,E2 -22779.53} C_VEL
LIN {X 0,Y 170.337,Z 440.875,A -85,B 0,C 180,E1 -22781.906,E2 -22781.906} C_VEL
LIN {X 0,Y 171.099,Z 434.673,A -85,B 0,C 180,E1 -22784.268,E2 -22784.268} C_VEL
LIN {X 0,Y 172.021,Z 428.164,A -85,B 0,C 180,E1 -22786.313,E2 -22786.313} C_VEL
LIN {X 0,Y 173.198,Z 420.318,A -85,B 0,C 180,E1 -22788.33,E2 -22788.33} C_VEL
LIN {X 0,Y 174.463,Z 410.557,A -85,B 0,C 180,E1 -22790.331,E2 -22790.331} C_VEL
LIN {X 0,Y 175.955,Z 399.521,A -85,B 0,C 180,E1 -22791.991,E2 -22791.991} C_VEL
LIN {X 0,Y 176.894,Z 389.353,A -85,B 0,C 180,E1 -22793.1,E2 -22793.1} C_VEL
LIN {X 0,Y 177.56,Z 379.651,A -85,B 0,C 180,E1 -22793.833,E2 -22793.833} C_VEL
LIN {X 0,Y 178.411,Z 355.968,A -85,B 0,C 180,E1 -22795.036,E2 -22795.036} C_VEL
LIN {X 0,Y 174.446,Z 307.152,A -85,B 0,C 180,E1 -22797.938,E2 -22797.938} C_VEL
LIN {X 0,Y 173.32,Z 302.745,A -85,B 0,C 180,E1 -22798.302,E2 -22798.302} C_VEL
LIN {X 0,Y 171.549,Z 293.931,A -85,B 0,C 180,E1 -22803.314,E2 -22803.314} C_VEL
LIN {X 0,Y 171.384,Z 293.948,A -85,B 0,C 180,E1 -22808.816,E2 -22808.816} C_VEL
LIN {X 0,Y 171.325,Z 293.953,A -85,B 0,C 180,E1 -22814.216,E2 -22814.216} C_VEL
LIN {X 0,Y 171.337,Z 293.954,A -85,B 0,C 180,E1 -22818.98,E2 -22818.98} C_VEL
LIN {X 0,Y 171.388,Z 293.945,A -85,B 0,C 180,E1 -22822.039,E2 -22822.039} C_VEL
LIN {X 0,Y 171.4,Z 293.946,A -85,B 0,C 180,E1 -22825.091,E2 -22825.091} C_VEL
LIN {X 0,Y 171.45,Z 293.936,A -85,B 0,C 180,E1 -22830.533,E2 -22830.533} C_VEL
LIN {X 0,Y 171.459,Z 293.939,A -85,B 0,C 180,E1 -22835.8,E2 -22835.8} C_VEL
LIN {X 0,Y 171.58,Z 293.922,A -85,B 0,C 180,E1 -22840.87,E2 -22840.87} C_VEL
LIN {X 0,Y 171.575,Z 293.922,A -85,B 0,C 180,E1 -22845.771,E2 -22845.771} C_VEL
LIN {X 0,Y 171.848,Z 293.89,A -85,B 0,C 180,E1 -22850.583,E2 -22850.583} C_VEL
LIN {X 0,Y 171.814,Z 293.891,A -85,B 0,C 180,E1 -22855.305,E2 -22855.305} C_VEL
LIN {X 0,Y 172.331,Z 293.831,A -85,B 0,C 180,E1 -22859.998,E2 -22859.998} C_VEL
LIN {X 0,Y 171.82,Z 293.89,A -85,B 0,C 180,E1 -22864.69,E2 -22864.69} C_VEL
LIN {X 0,Y 171.889,Z 293.887,A -85,B 0,C 180,E1 -22869.411,E2 -22869.411} C_VEL
LIN {X 0,Y 171.578,Z 293.923,A -85,B 0,C 180,E1 -22874.225,E2 -22874.225} C_VEL
LIN {X 0,Y 171.57,Z 293.923,A -85,B 0,C 180,E1 -22879.586,E2 -22879.586} C_VEL
LIN {X 0,Y 171.466,Z 293.94,A -85,B 0,C 180,E1 -22885.615,E2 -22885.615} C_VEL
LIN {X 0,Y 171.438,Z 293.939,A -85,B 0,C 180,E1 -22890.585,E2 -22890.585} C_VEL
LIN {X 0,Y 171.403,Z 293.945,A -85,B 0,C 180,E1 -22895.03,E2 -22895.03} C_VEL
LIN {X 0,Y 171.396,Z 293.943,A -85,B 0,C 180,E1 -22898.824,E2 -22898.824} C_VEL
LIN {X 0,Y 171.434,Z 293.94,A -85,B 0,C 180,E1 -22904.177,E2 -22904.177} C_VEL
LIN {X 0,Y 171.414,Z 293.943,A -85,B 0,C 180,E1 -22909.005,E2 -22909.005} C_VEL
LIN {X 0,Y 171.432,Z 293.942,A -85,B 0,C 180,E1 -22912.053,E2 -22912.053} C_VEL
LIN {X 0,Y 171.414,Z 293.946,A -85,B 0,C 180,E1 -22917.792,E2 -22917.792} C_VEL
LIN {X 0,Y 171.443,Z 293.94,A -85,B 0,C 180,E1 -22920.533,E2 -22920.533} C_VEL
LIN {X 0,Y 171.452,Z 293.941,A -85,B 0,C 180,E1 -22925.801,E2 -22925.801} C_VEL
LIN {X 0,Y 171.573,Z 293.921,A -85,B 0,C 180,E1 -22930.871,E2 -22930.871} C_VEL
LIN {X 0,Y 171.603,Z 293.923,A -85,B 0,C 180,E1 -22935.775,E2 -22935.775} C_VEL
LIN {X 0,Y 171.867,Z 293.884,A -85,B 0,C 180,E1 -22940.586,E2 -22940.586} C_VEL
LIN {X 0,Y 171.814,Z 293.895,A -85,B 0,C 180,E1 -22945.307,E2 -22945.307} C_VEL
LIN {X 0,Y 172.326,Z 293.83,A -85,B 0,C 180,E1 -22949.999,E2 -22949.999} C_VEL
LIN {X 0,Y 171.813,Z 293.893,A -85,B 0,C 180,E1 -22954.692,E2 -22954.692} C_VEL
LIN {X 0,Y 171.881,Z 293.885,A -85,B 0,C 180,E1 -22959.413,E2 -22959.413} C_VEL
LIN {X 0,Y 171.602,Z 293.919,A -85,B 0,C 180,E1 -22964.224,E2 -22964.224} C_VEL
LIN {X 0,Y 171.531,Z 293.93,A -85,B 0,C 180,E1 -22969.556,E2 -22969.556} C_VEL
LIN {X 0,Y 171.5,Z 293.934,A -85,B 0,C 180,E1 -22971.152,E2 -22971.152} C_VEL
LIN {X 0,Y 179.613,Z 317.749,A -85,B 0,C 180,E1 -22973.185,E2 -22973.185} C_VEL
LIN {X 0,Y 177.725,Z 361.553,A -85,B 0,C 180,E1 -22975.354,E2 -22975.354} C_VEL
LIN {X 0,Y 177.156,Z 371.849,A -85,B 0,C 180,E1 -22976.188,E2 -22976.188} C_VEL
LIN {X 0,Y 176.002,Z 384.057,A -85,B 0,C 180,E1 -22977.657,E2 -22977.657} C_VEL
LIN {X 0,Y 175.066,Z 392.985,A -85,B 0,C 180,E1 -22979.126,E2 -22979.126} C_VEL
LIN {X 0,Y 173.902,Z 402.073,A -85,B 0,C 180,E1 -22981.014,E2 -22981.014} C_VEL
LIN {X 0,Y 172.509,Z 411.104,A -85,B 0,C 180,E1 -22983.365,E2 -22983.365} C_VEL
LIN {X 0,Y 171.316,Z 419.366,A -85,B 0,C 180,E1 -22986.134,E2 -22986.134} C_VEL
LIN {X 0,Y 170.33,Z 426.256,A -85,B 0,C 180,E1 -22989.076,E2 -22989.076} C_VEL
LIN {X 0,Y 169.71,Z 431.395,A -85,B 0,C 180,E1 -22991.809,E2 -22991.809} C_VEL
LIN {X 0,Y 169.138,Z 436.032,A -85,B 0,C 180,E1 -22994.939,E2 -22994.939} C_VEL
LIN {X 0,Y 168.935,Z 439.98,A -85,B 0,C 180,E1 -22998.487,E2 -22998.487} C_VEL
LIN {X 0,Y 169.236,Z 442.671,A -85,B 0,C 180,E1 -23002.092,E2 -23002.092} C_VEL
LIN {X 0,Y 170.072,Z 444.127,A -85,B 0,C 180,E1 -23005.736,E2 -23005.736} C_VEL
LIN {X 0,Y 170.77,Z 444.494,A -85,B 0,C 180,E1 -23007.658,E2 -23007.658} C_VEL
LIN {X 0,Y 172.112,Z 444.32,A -85,B 0,C 180,E1 -23010.662,E2 -23010.662} C_VEL
LIN {X 0,Y 173.897,Z 443.317,A -85,B 0,C 180,E1 -23013.607,E2 -23013.607} C_VEL
LIN {X 0,Y 176.13,Z 441.411,A -85,B 0,C 180,E1 -23016.596,E2 -23016.596} C_VEL
LIN {X 0,Y 179.39,Z 437.78,A -85,B 0,C 180,E1 -23020.09,E2 -23020.09} C_VEL
LIN {X 0,Y 182.47,Z 433.757,A -85,B 0,C 180,E1 -23022.804,E2 -23022.804} C_VEL
LIN {X 0,Y 185.626,Z 429.159,A -85,B 0,C 180,E1 -23025.154,E2 -23025.154} C_VEL
LIN {X 0,Y 188.448,Z 424.498,A -85,B 0,C 180,E1 -23027.072,E2 -23027.072} C_VEL
LIN {X 0,Y 191.922,Z 418.024,A -85,B 0,C 180,E1 -23029.185,E2 -23029.185} C_VEL
LIN {X 0,Y 195.052,Z 411.397,A -85,B 0,C 180,E1 -23030.932,E2 -23030.932} C_VEL
LIN {X 0,Y 197.769,Z 404.802,A -85,B 0,C 180,E1 -23032.356,E2 -23032.356} C_VEL
LIN {X 0,Y 200.721,Z 396.535,A -85,B 0,C 180,E1 -23033.781,E2 -23033.781} C_VEL
LIN {X 0,Y 203.554,Z 386.915,A -85,B 0,C 180,E1 -23035.071,E2 -23035.071} C_VEL
LIN {X 0,Y 206.064,Z 375.094,A -85,B 0,C 180,E1 -23036.251,E2 -23036.251} C_VEL
LIN {X 0,Y 207.582,Z 364.747,A -85,B 0,C 180,E1 -23036.939,E2 -23036.939} C_VEL
LIN {X 0,Y 209.368,Z 345.672,A -85,B 0,C 180,E1 -23037.788,E2 -23037.788} C_VEL
LIN {X 0,Y 205.553,Z 337.923,A -85,B 0,C 180,E1 -23039.966,E2 -23039.966} C_VEL
LIN {X 0,Y 199.812,Z 328.185,A -85,B 0,C 180,E1 -23043.665,E2 -23043.665} C_VEL
LIN {X 0,Y 198.262,Z 325.838,A -85,B 0,C 180,E1 -23044.799,E2 -23044.799} C_VEL
LIN {X 0,Y 195.289,Z 321.819,A -85,B 0,C 180,E1 -23047.17,E2 -23047.17} C_VEL
LIN {X 0,Y 192.793,Z 318.641,A -85,B 0,C 180,E1 -23049.502,E2 -23049.502} C_VEL
LIN {X 0,Y 192.051,Z 317.164,A -85,B 0,C 180,E1 -23050.338,E2 -23050.338} C_VEL
LIN {X 0,Y 189.283,Z 314.56,A -85,B 0,C 180,E1 -23053.694,E2 -23053.694} C_VEL
LIN {X 0,Y 188.124,Z 311.996,A -85,B 0,C 180,E1 -23055.867,E2 -23055.867} C_VEL
LIN {X 0,Y 185.891,Z 310.798,A -85,B 0,C 180,E1 -23062.216,E2 -23062.216} C_VEL
LIN {X 0,Y 186.052,Z 310.982,A -85,B 0,C 180,E1 -23066.957,E2 -23066.957} C_VEL
LIN {X 0,Y 186.561,Z 311.662,A -85,B 0,C 180,E1 -23069.073,E2 -23069.073} C_VEL
LIN {X 0,Y 189.115,Z 315.41,A -85,B 0,C 180,E1 -23074.363,E2 -23074.363} C_VEL
LIN {X 0,Y 193.301,Z 322.417,A -85,B 0,C 180,E1 -23079.521,E2 -23079.521} C_VEL
LIN {X 0,Y 196.761,Z 328.68,A -85,B 0,C 180,E1 -23082.688,E2 -23082.688} C_VEL
LIN {X 0,Y 199.678,Z 334.305,A -85,B 0,C 180,E1 -23084.971,E2 -23084.971} C_VEL
LIN {X 0,Y 202.433,Z 339.934,A -85,B 0,C 180,E1 -23086.872,E2 -23086.872} C_VEL
LIN {X 0,Y 206.188,Z 349.087,A -85,B 0,C 180,E1 -23089.321,E2 -23089.321} C_VEL
LIN {X 0,Y 207.326,Z 352.705,A -85,B 0,C 180,E1 -23090.05,E2 -23090.05} C_VEL
LIN {X 0,Y 207.952,Z 365.84,A -85,B 0,C 180,E1 -23091.272,E2 -23091.272} C_VEL
LIN {X 0,Y 206.069,Z 382.212,A -85,B 0,C 180,E1 -23092.002,E2 -23092.002} C_VEL
LIN {X 0,Y 203.848,Z 393.06,A -85,B 0,C 180,E1 -23092.766,E2 -23092.766} C_VEL
LIN {X 0,Y 201.498,Z 401.981,A -85,B 0,C 180,E1 -23093.636,E2 -23093.636} C_VEL
LIN {X 0,Y 198.338,Z 411.543,A -85,B 0,C 180,E1 -23094.845,E2 -23094.845} C_VEL
LIN {X 0,Y 194.383,Z 421.613,A -85,B 0,C 180,E1 -23096.54,E2 -23096.54} C_VEL
LIN {X 0,Y 190.766,Z 429.574,A -85,B 0,C 180,E1 -23098.334,E2 -23098.334} C_VEL
LIN {X 0,Y 187.397,Z 436.178,A -85,B 0,C 180,E1 -23100.205,E2 -23100.205} C_VEL
LIN {X 0,Y 184.583,Z 441.18,A -85,B 0,C 180,E1 -23101.929,E2 -23101.929} C_VEL
LIN {X 0,Y 181.941,Z 444.625,A -85,B 0,C 180,E1 -23103.21,E2 -23103.21} C_VEL
LIN {X 0,Y 176.159,Z 449.637,A -85,B 0,C 180,E1 -23105.243,E2 -23105.243} C_VEL
LIN {X 0,Y 170.548,Z 453.776,A -85,B 0,C 180,E1 -23107.554,E2 -23107.554} C_VEL
LIN {X 0,Y 168.231,Z 455.739,A -85,B 0,C 180,E1 -23109.24,E2 -23109.24} C_VEL
LIN {X 0,Y 165.565,Z 458.687,A -85,B 0,C 180,E1 -23112.715,E2 -23112.715} C_VEL
LIN {X 0,Y 164.28,Z 459.997,A -85,B 0,C 180,E1 -23115.128,E2 -23115.128} C_VEL
LIN {X 0,Y 163.247,Z 460.871,A -85,B 0,C 180,E1 -23117.57,E2 -23117.57} C_VEL
LIN {X 0,Y 162.584,Z 461.305,A -85,B 0,C 180,E1 -23120.044,E2 -23120.044} C_VEL
LIN {X 0,Y 162.218,Z 461.162,A -85,B 0,C 180,E1 -23122.533,E2 -23122.533} C_VEL
LIN {X 0,Y 162.173,Z 460.423,A -85,B 0,C 180,E1 -23125.391,E2 -23125.391} C_VEL
LIN {X 0,Y 162.274,Z 459.459,A -85,B 0,C 180,E1 -23127.518,E2 -23127.518} C_VEL
LIN {X 0,Y 162.385,Z 457.87,A -85,B 0,C 180,E1 -23130.001,E2 -23130.001} C_VEL
LIN {X 0,Y 162.41,Z 455.64,A -85,B 0,C 180,E1 -23132.481,E2 -23132.481} C_VEL
LIN {X 0,Y 162.442,Z 450.987,A -85,B 0,C 180,E1 -23136.209,E2 -23136.209} C_VEL
LIN {X 0,Y 162.713,Z 445.83,A -85,B 0,C 180,E1 -23139.322,E2 -23139.322} C_VEL
LIN {X 0,Y 163.213,Z 440.744,A -85,B 0,C 180,E1 -23141.803,E2 -23141.803} C_VEL
LIN {X 0,Y 163.981,Z 434.598,A -85,B 0,C 180,E1 -23144.267,E2 -23144.267} C_VEL
LIN {X 0,Y 165.077,Z 427.131,A -85,B 0,C 180,E1 -23146.701,E2 -23146.701} C_VEL
LIN {X 0,Y 166.287,Z 419.156,A -85,B 0,C 180,E1 -23148.8,E2 -23148.8} C_VEL
LIN {X 0,Y 167.616,Z 409.196,A -85,B 0,C 180,E1 -23150.879,E2 -23150.879} C_VEL
LIN {X 0,Y 169.017,Z 398.831,A -85,B 0,C 180,E1 -23152.46,E2 -23152.46} C_VEL
LIN {X 0,Y 169.937,Z 389.35,A -85,B 0,C 180,E1 -23153.538,E2 -23153.538} C_VEL
LIN {X 0,Y 170.636,Z 379.483,A -85,B 0,C 180,E1 -23154.322,E2 -23154.322} C_VEL
LIN {X 0,Y 171.453,Z 355.502,A -85,B 0,C 180,E1 -23155.601,E2 -23155.601} C_VEL
LIN {X 0,Y 167.701,Z 308.696,A -85,B 0,C 180,E1 -23158.513,E2 -23158.513} C_VEL
LIN {X 0,Y 165.992,Z 302.306,A -85,B 0,C 180,E1 -23159.071,E2 -23159.071} C_VEL
LIN {X 0,Y 164.486,Z 294.81,A -85,B 0,C 180,E1 -23163.601,E2 -23163.601} C_VEL
LIN {X 0,Y 164.309,Z 294.831,A -85,B 0,C 180,E1 -23169.651,E2 -23169.651} C_VEL
LIN {X 0,Y 164.283,Z 294.829,A -85,B 0,C 180,E1 -23173.341,E2 -23173.341} C_VEL
LIN {X 0,Y 164.266,Z 294.835,A -85,B 0,C 180,E1 -23176.798,E2 -23176.798} C_VEL
LIN {X 0,Y 164.297,Z 294.827,A -85,B 0,C 180,E1 -23180.351,E2 -23180.351} C_VEL
LIN {X 0,Y 164.332,Z 294.826,A -85,B 0,C 180,E1 -23184.348,E2 -23184.348} C_VEL
LIN {X 0,Y 164.391,Z 294.817,A -85,B 0,C 180,E1 -23189.133,E2 -23189.133} C_VEL
LIN {X 0,Y 164.418,Z 294.816,A -85,B 0,C 180,E1 -23194.692,E2 -23194.692} C_VEL
LIN {X 0,Y 164.486,Z 294.807,A -85,B 0,C 180,E1 -23200.049,E2 -23200.049} C_VEL
LIN {X 0,Y 164.523,Z 294.802,A -85,B 0,C 180,E1 -23205.147,E2 -23205.147} C_VEL
LIN {X 0,Y 164.768,Z 294.773,A -85,B 0,C 180,E1 -23210.174,E2 -23210.174} C_VEL
LIN {X 0,Y 164.83,Z 294.764,A -85,B 0,C 180,E1 -23212.649,E2 -23212.649} C_VEL
LIN {X 0,Y 165.046,Z 294.737,A -85,B 0,C 180,E1 -23217.557,E2 -23217.557} C_VEL
LIN {X 0,Y 165.294,Z 294.707,A -85,B 0,C 180,E1 -23219.998,E2 -23219.998} C_VEL
LIN {X 0,Y 164.77,Z 294.768,A -85,B 0,C 180,E1 -23224.892,E2 -23224.892} C_VEL
LIN {X 0,Y 164.852,Z 294.762,A -85,B 0,C 180,E1 -23227.346,E2 -23227.346} C_VEL
LIN {X 0,Y 164.741,Z 294.774,A -85,B 0,C 180,E1 -23231.129,E2 -23231.129} C_VEL
LIN {X 0,Y 164.501,Z 294.807,A -85,B 0,C 180,E1 -23237.399,E2 -23237.399} C_VEL
LIN {X 0,Y 164.5,Z 294.801,A -85,B 0,C 180,E1 -23239.983,E2 -23239.983} C_VEL
LIN {X 0,Y 164.39,Z 294.819,A -85,B 0,C 180,E1 -23246.132,E2 -23246.132} C_VEL
LIN {X 0,Y 164.372,Z 294.82,A -85,B 0,C 180,E1 -23251.226,E2 -23251.226} C_VEL
LIN {X 0,Y 164.313,Z 294.825,A -85,B 0,C 180,E1 -23256.782,E2 -23256.782} C_VEL
LIN {X 0,Y 164.333,Z 294.827,A -85,B 0,C 180,E1 -23259.901,E2 -23259.901} C_VEL
LIN {X 0,Y 164.368,Z 294.823,A -85,B 0,C 180,E1 -23263.375,E2 -23263.375} C_VEL
LIN {X 0,Y 164.379,Z 294.816,A -85,B 0,C 180,E1 -23266.837,E2 -23266.837} C_VEL
LIN {X 0,Y 164.365,Z 294.823,A -85,B 0,C 180,E1 -23270.319,E2 -23270.319} C_VEL
LIN {X 0,Y 164.339,Z 294.82,A -85,B 0,C 180,E1 -23274.34,E2 -23274.34} C_VEL
LIN {X 0,Y 164.385,Z 294.82,A -85,B 0,C 180,E1 -23279.134,E2 -23279.134} C_VEL
LIN {X 0,Y 164.411,Z 294.814,A -85,B 0,C 180,E1 -23284.693,E2 -23284.693} C_VEL
LIN {X 0,Y 164.479,Z 294.806,A -85,B 0,C 180,E1 -23290.05,E2 -23290.05} C_VEL
LIN {X 0,Y 164.547,Z 294.8,A -85,B 0,C 180,E1 -23295.151,E2 -23295.151} C_VEL
LIN {X 0,Y 164.792,Z 294.766,A -85,B 0,C 180,E1 -23300.177,E2 -23300.177} C_VEL
LIN {X 0,Y 164.84,Z 294.762,A -85,B 0,C 180,E1 -23302.651,E2 -23302.651} C_VEL
LIN {X 0,Y 165.042,Z 294.737,A -85,B 0,C 180,E1 -23307.559,E2 -23307.559} C_VEL
LIN {X 0,Y 165.288,Z 294.706,A -85,B 0,C 180,E1 -23309.999,E2 -23309.999} C_VEL
LIN {X 0,Y 164.763,Z 294.772,A -85,B 0,C 180,E1 -23314.893,E2 -23314.893} C_VEL
LIN {X 0,Y 164.843,Z 294.758,A -85,B 0,C 180,E1 -23317.348,E2 -23317.348} C_VEL
LIN {X 0,Y 164.747,Z 294.775,A -85,B 0,C 180,E1 -23321.151,E2 -23321.151} C_VEL
LIN {X 0,Y 164.493,Z 294.807,A -85,B 0,C 180,E1 -23327.401,E2 -23327.401} C_VEL
LIN {X 0,Y 164.46,Z 294.816,A -85,B 0,C 180,E1 -23330.478,E2 -23330.478} C_VEL
LIN {X 0,Y 172.789,Z 319.159,A -85,B 0,C 180,E1 -23332.647,E2 -23332.647} C_VEL
LIN {X 0,Y 170.829,Z 362.552,A -85,B 0,C 180,E1 -23334.889,E2 -23334.889} C_VEL
LIN {X 0,Y 170.027,Z 374.154,A -85,B 0,C 180,E1 -23335.896,E2 -23335.896} C_VEL
LIN {X 0,Y 169.046,Z 384.287,A -85,B 0,C 180,E1 -23337.213,E2 -23337.213} C_VEL
LIN {X 0,Y 167.982,Z 393.916,A -85,B 0,C 180,E1 -23338.874,E2 -23338.874} C_VEL
LIN {X 0,Y 167.139,Z 400.638,A -85,B 0,C 180,E1 -23340.302,E2 -23340.302} C_VEL
LIN {X 0,Y 165.968,Z 407.813,A -85,B 0,C 180,E1 -23342.127,E2 -23342.127} C_VEL
LIN {X 0,Y 165.005,Z 414.223,A -85,B 0,C 180,E1 -23344.089,E2 -23344.089} C_VEL
LIN {X 0,Y 164.166,Z 420,A -85,B 0,C 180,E1 -23346.191,E2 -23346.191} C_VEL
LIN {X 0,Y 163.177,Z 426.662,A -85,B 0,C 180,E1 -23349.176,E2 -23349.176} C_VEL
LIN {X 0,Y 162.675,Z 430.933,A -85,B 0,C 180,E1 -23351.495,E2 -23351.495} C_VEL
LIN {X 0,Y 162.03,Z 436.011,A -85,B 0,C 180,E1 -23354.965,E2 -23354.965} C_VEL
LIN {X 0,Y 161.849,Z 438.99,A -85,B 0,C 180,E1 -23357.575,E2 -23357.575} C_VEL
LIN {X 0,Y 161.881,Z 440.732,A -85,B 0,C 180,E1 -23359.37,E2 -23359.37} C_VEL
LIN {X 0,Y 162.215,Z 443.042,A -85,B 0,C 180,E1 -23362.663,E2 -23362.663} C_VEL
LIN {X 0,Y 163.013,Z 444.432,A -85,B 0,C 180,E1 -23365.915,E2 -23365.915} C_VEL
LIN {X 0,Y 164.215,Z 444.956,A -85,B 0,C 180,E1 -23369.101,E2 -23369.101} C_VEL
LIN {X 0,Y 166.093,Z 444.492,A -85,B 0,C 180,E1 -23372.693,E2 -23372.693} C_VEL
LIN {X 0,Y 168.69,Z 442.792,A -85,B 0,C 180,E1 -23376.425,E2 -23376.425} C_VEL
LIN {X 0,Y 170.19,Z 441.591,A -85,B 0,C 180,E1 -23378.185,E2 -23378.185} C_VEL
LIN {X 0,Y 173.008,Z 438.752,A -85,B 0,C 180,E1 -23381.038,E2 -23381.038} C_VEL
LIN {X 0,Y 176.185,Z 434.946,A -85,B 0,C 180,E1 -23383.788,E2 -23383.788} C_VEL
LIN {X 0,Y 179.89,Z 429.987,A -85,B 0,C 180,E1 -23386.445,E2 -23386.445} C_VEL
LIN {X 0,Y 182.97,Z 425.29,A -85,B 0,C 180,E1 -23388.453,E2 -23388.453} C_VEL
LIN {X 0,Y 186.788,Z 418.625,A -85,B 0,C 180,E1 -23390.692,E2 -23390.692} C_VEL
LIN {X 0,Y 189.897,Z 412.453,A -85,B 0,C 180,E1 -23392.353,E2 -23392.353} C_VEL
LIN {X 0,Y 193.188,Z 404.885,A -85,B 0,C 180,E1 -23393.999,E2 -23393.999} C_VEL
LIN {X 0,Y 196.205,Z 396.821,A -85,B 0,C 180,E1 -23395.38,E2 -23395.38} C_VEL
LIN {X 0,Y 199.134,Z 387.3,A -85,B 0,C 180,E1 -23396.655,E2 -23396.655} C_VEL
LIN {X 0,Y 201.769,Z 375.612,A -85,B 0,C 180,E1 -23397.825,E2 -23397.825} C_VEL
LIN {X 0,Y 203.399,Z 365.118,A -85,B 0,C 180,E1 -23398.531,E2 -23398.531} C_VEL
LIN {X 0,Y 205.05,Z 348.84,A -85,B 0,C 180,E1 -23399.271,E2 -23399.271} C_VEL
LIN {X 0,Y 202.068,Z 342.818,A -85,B 0,C 180,E1 -23401.116,E2 -23401.116} C_VEL
LIN {X 0,Y 197.036,Z 333.784,A -85,B 0,C 180,E1 -23404.662,E2 -23404.662} C_VEL
LIN {X 0,Y 195.258,Z 331.272,A -85,B 0,C 180,E1 -23406.025,E2 -23406.025} C_VEL
LIN {X 0,Y 193.252,Z 328.331,A -85,B 0,C 180,E1 -23407.808,E2 -23407.808} C_VEL
LIN {X 0,Y 190.659,Z 324.678,A -85,B 0,C 180,E1 -23410.414,E2 -23410.414} C_VEL
LIN {X 0,Y 190.119,Z 323.72,A -85,B 0,C 180,E1 -23411.098,E2 -23411.098} C_VEL
LIN {X 0,Y 187.723,Z 321.258,A -85,B 0,C 180,E1 -23414.224,E2 -23414.224} C_VEL
LIN {X 0,Y 186.769,Z 318.955,A -85,B 0,C 180,E1 -23416.204,E2 -23416.204} C_VEL
LIN {X 0,Y 184.724,Z 317.798,A -85,B 0,C 180,E1 -23422.364,E2 -23422.364} C_VEL
LIN {X 0,Y 185.046,Z 318.092,A -85,B 0,C 180,E1 -23427.666,E2 -23427.666} C_VEL
LIN {X 0,Y 187.018,Z 321.305,A -85,B 0,C 180,E1 -23432.938,E2 -23432.938} C_VEL
LIN {X 0,Y 187.848,Z 322.864,A -85,B 0,C 180,E1 -23434.344,E2 -23434.344} C_VEL
LIN {X 0,Y 191.252,Z 328.711,A -85,B 0,C 180,E1 -23438.753,E2 -23438.753} C_VEL
LIN {X 0,Y 194.292,Z 334.664,A -85,B 0,C 180,E1 -23441.817,E2 -23441.817} C_VEL
LIN {X 0,Y 197.147,Z 340.45,A -85,B 0,C 180,E1 -23444.189,E2 -23444.189} C_VEL
LIN {X 0,Y 199.969,Z 346.694,A -85,B 0,C 180,E1 -23446.309,E2 -23446.309} C_VEL
LIN {X 0,Y 203.287,Z 355.614,A -85,B 0,C 180,E1 -23448.621,E2 -23448.621} C_VEL
LIN {X 0,Y 203.658,Z 366.304,A -85,B 0,C 180,E1 -23449.67,E2 -23449.67} C_VEL
LIN {X 0,Y 201.768,Z 382.151,A -85,B 0,C 180,E1 -23450.414,E2 -23450.414} C_VEL
LIN {X 0,Y 199.783,Z 391.694,A -85,B 0,C 180,E1 -23451.076,E2 -23451.076} C_VEL
LIN {X 0,Y 197.34,Z 400.655,A -85,B 0,C 180,E1 -23451.909,E2 -23451.909} C_VEL
LIN {X 0,Y 194.304,Z 409.76,A -85,B 0,C 180,E1 -23453.036,E2 -23453.036} C_VEL
LIN {X 0,Y 191.143,Z 417.695,A -85,B 0,C 180,E1 -23454.291,E2 -23454.291} C_VEL
LIN {X 0,Y 187.613,Z 425.349,A -85,B 0,C 180,E1 -23455.814,E2 -23455.814} C_VEL
LIN {X 0,Y 183.046,Z 434.257,A -85,B 0,C 180,E1 -23458.136,E2 -23458.136} C_VEL
LIN {X 0,Y 178.488,Z 441.806,A -85,B 0,C 180,E1 -23460.814,E2 -23460.814} C_VEL
LIN {X 0,Y 174.348,Z 447.916,A -85,B 0,C 180,E1 -23463.679,E2 -23463.679} C_VEL
LIN {X 0,Y 171.652,Z 451.504,A -85,B 0,C 180,E1 -23465.832,E2 -23465.832} C_VEL
LIN {X 0,Y 168.231,Z 455.739,A -85,B 0,C 180,E1 -23469.24,E2 -23469.24} C_VEL
LIN {X 0,Y 166.058,Z 457.516,A -85,B 0,C 180,E1 -23471.032,E2 -23471.032} C_VEL
LIN {X 0,Y 163.224,Z 458.906,A -85,B 0,C 180,E1 -23472.792,E2 -23472.792} C_VEL
LIN {X 0,Y 158.431,Z 460.361,A -85,B 0,C 180,E1 -23475.848,E2 -23475.848} C_VEL
LIN {X 0,Y 155.92,Z 460.832,A -85,B 0,C 180,E1 -23478.563,E2 -23478.563} C_VEL
LIN {X 0,Y 155.658,Z 460.802,A -85,B 0,C 180,E1 -23479.279,E2 -23479.279} C_VEL
LIN {X 0,Y 155.171,Z 460.668,A -85,B 0,C 180,E1 -23482.192,E2 -23482.192} C_VEL
LIN {X 0,Y 155.107,Z 459.713,A -85,B 0,C 180,E1 -23485.459,E2 -23485.459} C_VEL
LIN {X 0,Y 155.212,Z 458.693,A -85,B 0,C 180,E1 -23487.405,E2 -23487.405} C_VEL
LIN {X 0,Y 155.335,Z 456.952,A -85,B 0,C 180,E1 -23490.001,E2 -23490.001} C_VEL
LIN {X 0,Y 155.374,Z 453.562,A -85,B 0,C 180,E1 -23493.516,E2 -23493.516} C_VEL
LIN {X 0,Y 155.401,Z 449.722,A -85,B 0,C 180,E1 -23496.491,E2 -23496.491} C_VEL
LIN {X 0,Y 155.731,Z 444.372,A -85,B 0,C 180,E1 -23499.744,E2 -23499.744} C_VEL
LIN {X 0,Y 156.455,Z 437.652,A -85,B 0,C 180,E1 -23502.98,E2 -23502.98} C_VEL
LIN {X 0,Y 157.653,Z 429.053,A -85,B 0,C 180,E1 -23506.178,E2 -23506.178} C_VEL
LIN {X 0,Y 158.83,Z 421.564,A -85,B 0,C 180,E1 -23508.377,E2 -23508.377} C_VEL
LIN {X 0,Y 159.952,Z 413.752,A -85,B 0,C 180,E1 -23510.244,E2 -23510.244} C_VEL
LIN {X 0,Y 161.035,Z 405.816,A -85,B 0,C 180,E1 -23511.775,E2 -23511.775} C_VEL
LIN {X 0,Y 162.225,Z 396.915,A -85,B 0,C 180,E1 -23513.117,E2 -23513.117} C_VEL
LIN {X 0,Y 163.094,Z 387.725,A -85,B 0,C 180,E1 -23514.166,E2 -23514.166} C_VEL
LIN {X 0,Y 163.887,Z 376.277,A -85,B 0,C 180,E1 -23515.054,E2 -23515.054} C_VEL
LIN {X 0,Y 164.575,Z 356.12,A -85,B 0,C 180,E1 -23516.146,E2 -23516.146} C_VEL
LIN {X 0,Y 160.919,Z 309.969,A -85,B 0,C 180,E1 -23519.131,E2 -23519.131} C_VEL
LIN {X 0,Y 158.689,Z 301.914,A -85,B 0,C 180,E1 -23519.875,E2 -23519.875} C_VEL
LIN {X 0,Y 157.438,Z 295.687,A -85,B 0,C 180,E1 -23523.725,E2 -23523.725} C_VEL
LIN {X 0,Y 157.251,Z 295.709,A -85,B 0,C 180,E1 -23528.734,E2 -23528.734} C_VEL
LIN {X 0,Y 157.181,Z 295.715,A -85,B 0,C 180,E1 -23534.321,E2 -23534.321} C_VEL
LIN {X 0,Y 157.201,Z 295.714,A -85,B 0,C 180,E1 -23539.465,E2 -23539.465} C_VEL
LIN {X 0,Y 157.281,Z 295.704,A -85,B 0,C 180,E1 -23544.484,E2 -23544.484} C_VEL
LIN {X 0,Y 157.295,Z 295.701,A -85,B 0,C 180,E1 -23548.095,E2 -23548.095} C_VEL
LIN {X 0,Y 157.324,Z 295.701,A -85,B 0,C 180,E1 -23553.464,E2 -23553.464} C_VEL
LIN {X 0,Y 157.395,Z 295.688,A -85,B 0,C 180,E1 -23559.666,E2 -23559.666} C_VEL
LIN {X 0,Y 157.453,Z 295.682,A -85,B 0,C 180,E1 -23564.464,E2 -23564.464} C_VEL
LIN {X 0,Y 157.69,Z 295.655,A -85,B 0,C 180,E1 -23569.729,E2 -23569.729} C_VEL
LIN {X 0,Y 157.767,Z 295.644,A -85,B 0,C 180,E1 -23572.318,E2 -23572.318} C_VEL
LIN {X 0,Y 158.256,Z 295.584,A -85,B 0,C 180,E1 -23579.998,E2 -23579.998} C_VEL
LIN {X 0,Y 157.808,Z 295.641,A -85,B 0,C 180,E1 -23587.676,E2 -23587.676} C_VEL
LIN {X 0,Y 157.671,Z 295.655,A -85,B 0,C 180,E1 -23591.299,E2 -23591.299} C_VEL
LIN {X 0,Y 157.461,Z 295.683,A -85,B 0,C 180,E1 -23595.531,E2 -23595.531} C_VEL
LIN {X 0,Y 157.382,Z 295.687,A -85,B 0,C 180,E1 -23600.929,E2 -23600.929} C_VEL
LIN {X 0,Y 157.311,Z 295.7,A -85,B 0,C 180,E1 -23606.683,E2 -23606.683} C_VEL
LIN {X 0,Y 157.274,Z 295.706,A -85,B 0,C 180,E1 -23612.425,E2 -23612.425} C_VEL
LIN {X 0,Y 157.281,Z 295.701,A -85,B 0,C 180,E1 -23616.456,E2 -23616.456} C_VEL
LIN {X 0,Y 157.271,Z 295.707,A -85,B 0,C 180,E1 -23622.087,E2 -23622.087} C_VEL
LIN {X 0,Y 157.296,Z 295.7,A -85,B 0,C 180,E1 -23625.63,E2 -23625.63} C_VEL
LIN {X 0,Y 157.282,Z 295.706,A -85,B 0,C 180,E1 -23631.275,E2 -23631.275} C_VEL
LIN {X 0,Y 157.286,Z 295.698,A -85,B 0,C 180,E1 -23634.488,E2 -23634.488} C_VEL
LIN {X 0,Y 157.289,Z 295.705,A -85,B 0,C 180,E1 -23638.094,E2 -23638.094} C_VEL
LIN {X 0,Y 157.316,Z 295.696,A -85,B 0,C 180,E1 -23643.465,E2 -23643.465} C_VEL
LIN {X 0,Y 157.388,Z 295.691,A -85,B 0,C 180,E1 -23649.666,E2 -23649.666} C_VEL
LIN {X 0,Y 157.472,Z 295.681,A -85,B 0,C 180,E1 -23654.467,E2 -23654.467} C_VEL
LIN {X 0,Y 157.72,Z 295.647,A -85,B 0,C 180,E1 -23659.732,E2 -23659.732} C_VEL
LIN {X 0,Y 157.797,Z 295.64,A -85,B 0,C 180,E1 -23662.321,E2 -23662.321} C_VEL
LIN {X 0,Y 158.251,Z 295.582,A -85,B 0,C 180,E1 -23669.999,E2 -23669.999} C_VEL
LIN {X 0,Y 157.801,Z 295.636,A -85,B 0,C 180,E1 -23677.678,E2 -23677.678} C_VEL
LIN {X 0,Y 157.676,Z 295.656,A -85,B 0,C 180,E1 -23681.321,E2 -23681.321} C_VEL
LIN {X 0,Y 157.469,Z 295.68,A -85,B 0,C 180,E1 -23685.532,E2 -23685.532} C_VEL
LIN {X 0,Y 157.444,Z 295.769,A -85,B 0,C 180,E1 -23689.764,E2 -23689.764} C_VEL
LIN {X 0,Y 165.807,Z 320.255,A -85,B 0,C 180,E1 -23692.055,E2 -23692.055} C_VEL
LIN {X 0,Y 163.908,Z 362.19,A -85,B 0,C 180,E1 -23694.322,E2 -23694.322} C_VEL
LIN {X 0,Y 163.208,Z 373.063,A -85,B 0,C 180,E1 -23695.278,E2 -23695.278} C_VEL
LIN {X 0,Y 162.083,Z 384.25,A -85,B 0,C 180,E1 -23696.734,E2 -23696.734} C_VEL
LIN {X 0,Y 161.088,Z 393.257,A -85,B 0,C 180,E1 -23698.323,E2 -23698.323} C_VEL
LIN {X 0,Y 160.065,Z 400.985,A -85,B 0,C 180,E1 -23700.014,E2 -23700.014} C_VEL
LIN {X 0,Y 158.787,Z 408.707,A -85,B 0,C 180,E1 -23702.08,E2 -23702.08} C_VEL
LIN {X 0,Y 157.721,Z 415.649,A -85,B 0,C 180,E1 -23704.351,E2 -23704.351} C_VEL
LIN {X 0,Y 156.774,Z 421.967,A -85,B 0,C 180,E1 -23706.859,E2 -23706.859} C_VEL
LIN {X 0,Y 156.077,Z 426.663,A -85,B 0,C 180,E1 -23709.078,E2 -23709.078} C_VEL
LIN {X 0,Y 155.568,Z 430.974,A -85,B 0,C 180,E1 -23711.48,E2 -23711.48} C_VEL
LIN {X 0,Y 155.012,Z 435.209,A -85,B 0,C 180,E1 -23714.356,E2 -23714.356} C_VEL
LIN {X 0,Y 154.77,Z 438.458,A -85,B 0,C 180,E1 -23717.071,E2 -23717.071} C_VEL
LIN {X 0,Y 154.867,Z 441.582,A -85,B 0,C 180,E1 -23720.559,E2 -23720.559} C_VEL
LIN {X 0,Y 155.471,Z 443.914,A -85,B 0,C 180,E1 -23724.454,E2 -23724.454} C_VEL
LIN {X 0,Y 156.75,Z 445.148,A -85,B 0,C 180,E1 -23728.413,E2 -23728.413} C_VEL
LIN {X 0,Y 158.669,Z 445.235,A -85,B 0,C 180,E1 -23732.355,E2 -23732.355} C_VEL
LIN {X 0,Y 161.832,Z 443.697,A -85,B 0,C 180,E1 -23736.995,E2 -23736.995} C_VEL
LIN {X 0,Y 164.514,Z 441.621,A -85,B 0,C 180,E1 -23740.018,E2 -23740.018} C_VEL
LIN {X 0,Y 168.455,Z 437.755,A -85,B 0,C 180,E1 -23743.646,E2 -23743.646} C_VEL
LIN {X 0,Y 172.299,Z 433.367,A -85,B 0,C 180,E1 -23746.514,E2 -23746.514} C_VEL
LIN {X 0,Y 176.904,Z 427.211,A -85,B 0,C 180,E1 -23749.503,E2 -23749.503} C_VEL
LIN {X 0,Y 181.701,Z 419.417,A -85,B 0,C 180,E1 -23752.223,E2 -23752.223} C_VEL
LIN {X 0,Y 185.197,Z 412.844,A -85,B 0,C 180,E1 -23754.012,E2 -23754.012} C_VEL
LIN {X 0,Y 188.234,Z 406.381,A -85,B 0,C 180,E1 -23755.451,E2 -23755.451} C_VEL
LIN {X 0,Y 191.675,Z 397.812,A -85,B 0,C 180,E1 -23756.965,E2 -23756.965} C_VEL
LIN {X 0,Y 194.629,Z 388.881,A -85,B 0,C 180,E1 -23758.191,E2 -23758.191} C_VEL
LIN {X 0,Y 197.441,Z 377.568,A -85,B 0,C 180,E1 -23759.4,E2 -23759.4} C_VEL
LIN {X 0,Y 199.393,Z 366.205,A -85,B 0,C 180,E1 -23760.166,E2 -23760.166} C_VEL
LIN {X 0,Y 200.871,Z 351.94,A -85,B 0,C 180,E1 -23760.861,E2 -23760.861} C_VEL
LIN {X 0,Y 198.324,Z 347.074,A -85,B 0,C 180,E1 -23762.566,E2 -23762.566} C_VEL
LIN {X 0,Y 194.522,Z 339.74,A -85,B 0,C 180,E1 -23765.521,E2 -23765.521} C_VEL
LIN {X 0,Y 191.471,Z 335.023,A -85,B 0,C 180,E1 -23768.254,E2 -23768.254} C_VEL
LIN {X 0,Y 188.846,Z 331.25,A -85,B 0,C 180,E1 -23771.062,E2 -23771.062} C_VEL
LIN {X 0,Y 188.243,Z 330.331,A -85,B 0,C 180,E1 -23771.843,E2 -23771.843} C_VEL
LIN {X 0,Y 185.921,Z 327.438,A -85,B 0,C 180,E1 -23775.26,E2 -23775.26} C_VEL
LIN {X 0,Y 185.302,Z 325.769,A -85,B 0,C 180,E1 -23776.778,E2 -23776.778} C_VEL
LIN {X 0,Y 183.485,Z 324.754,A -85,B 0,C 180,E1 -23783.185,E2 -23783.185} C_VEL
LIN {X 0,Y 183.986,Z 325.259,A -85,B 0,C 180,E1 -23788.117,E2 -23788.117} C_VEL
LIN {X 0,Y 185.927,Z 328.741,A -85,B 0,C 180,E1 -23793.156,E2 -23793.156} C_VEL
LIN {X 0,Y 189.295,Z 335.193,A -85,B 0,C 180,E1 -23798.061,E2 -23798.061} C_VEL
LIN {X 0,Y 191.998,Z 340.838,A -85,B 0,C 180,E1 -23800.992,E2 -23800.992} C_VEL
LIN {X 0,Y 194.751,Z 346.75,A -85,B 0,C 180,E1 -23803.462,E2 -23803.462} C_VEL
LIN {X 0,Y 197.247,Z 352.958,A -85,B 0,C 180,E1 -23805.531,E2 -23805.531} C_VEL
LIN {X 0,Y 199.483,Z 359.391,A -85,B 0,C 180,E1 -23807.23,E2 -23807.23} C_VEL
LIN {X 0,Y 199.6,Z 368.394,A -85,B 0,C 180,E1 -23808.082,E2 -23808.082} C_VEL
LIN {X 0,Y 197.657,Z 382.517,A -85,B 0,C 180,E1 -23808.763,E2 -23808.763} C_VEL
LIN {X 0,Y 195.525,Z 392.035,A -85,B 0,C 180,E1 -23809.437,E2 -23809.437} C_VEL
LIN {X 0,Y 192.733,Z 401.544,A -85,B 0,C 180,E1 -23810.349,E2 -23810.349} C_VEL
LIN {X 0,Y 189.329,Z 410.955,A -85,B 0,C 180,E1 -23811.556,E2 -23811.556} C_VEL
LIN {X 0,Y 184.913,Z 420.953,A -85,B 0,C 180,E1 -23813.231,E2 -23813.231} C_VEL
LIN {X 0,Y 180.907,Z 428.832,A -85,B 0,C 180,E1 -23815.041,E2 -23815.041} C_VEL
LIN {X 0,Y 177.126,Z 435.383,A -85,B 0,C 180,E1 -23816.938,E2 -23816.938} C_VEL
LIN {X 0,Y 172.768,Z 442.078,A -85,B 0,C 180,E1 -23819.438,E2 -23819.438} C_VEL
LIN {X 0,Y 169.564,Z 446.527,A -85,B 0,C 180,E1 -23821.535,E2 -23821.535} C_VEL
LIN {X 0,Y 165.228,Z 451.849,A -85,B 0,C 180,E1 -23824.828,E2 -23824.828} C_VEL
LIN {X 0,Y 162.747,Z 454.643,A -85,B 0,C 180,E1 -23827.131,E2 -23827.131} C_VEL
LIN {X 0,Y 160.597,Z 456.92,A -85,B 0,C 180,E1 -23829.508,E2 -23829.508} C_VEL
LIN {X 0,Y 158.78,Z 458.667,A -85,B 0,C 180,E1 -23831.952,E2 -23831.952} C_VEL
LIN {X 0,Y 157.408,Z 459.828,A -85,B 0,C 180,E1 -23834.462,E2 -23834.462} C_VEL
LIN {X 0,Y 155.658,Z 460.802,A -85,B 0,C 180,E1 -23839.279,E2 -23839.279} C_VEL
LIN {X 0,Y 154.634,Z 460.753,A -85,B 0,C 180,E1 -23841.425,E2 -23841.425} C_VEL
LIN {X 0,Y 152.93,Z 460.178,A -85,B 0,C 180,E1 -23843.534,E2 -23843.534} C_VEL
LIN {X 0,Y 149.324,Z 457.79,A -85,B 0,C 180,E1 -23847.778,E2 -23847.778} C_VEL
LIN {X 0,Y 148.267,Z 455.459,A -85,B 0,C 180,E1 -23850.706,E2 -23850.706} C_VEL
LIN {X 0,Y 148.33,Z 451.597,A -85,B 0,C 180,E1 -23854.479,E2 -23854.479} C_VEL
LIN {X 0,Y 148.464,Z 446.453,A -85,B 0,C 180,E1 -23858.165,E2 -23858.165} C_VEL
LIN {X 0,Y 149.021,Z 440.265,A -85,B 0,C 180,E1 -23861.563,E2 -23861.563} C_VEL
LIN {X 0,Y 149.758,Z 434.195,A -85,B 0,C 180,E1 -23864.264,E2 -23864.264} C_VEL
LIN {X 0,Y 150.879,Z 426.833,A -85,B 0,C 180,E1 -23866.926,E2 -23866.926} C_VEL
LIN {X 0,Y 152.127,Z 418.98,A -85,B 0,C 180,E1 -23869.218,E2 -23869.218} C_VEL
LIN {X 0,Y 153.477,Z 409.206,A -85,B 0,C 180,E1 -23871.49,E2 -23871.49} C_VEL
LIN {X 0,Y 155.095,Z 398.145,A -85,B 0,C 180,E1 -23873.36,E2 -23873.36} C_VEL
LIN {X 0,Y 156.049,Z 388.731,A -85,B 0,C 180,E1 -23874.531,E2 -23874.531} C_VEL
LIN {X 0,Y 156.812,Z 379.037,A -85,B 0,C 180,E1 -23875.377,E2 -23875.377} C_VEL
LIN {X 0,Y 157.66,Z 356.473,A -85,B 0,C 180,E1 -23876.699,E2 -23876.699} C_VEL
LIN {X 0,Y 154.17,Z 311.549,A -85,B 0,C 180,E1 -23879.755,E2 -23879.755} C_VEL
LIN {X 0,Y 151.383,Z 301.569,A -85,B 0,C 180,E1 -23880.709,E2 -23880.709} C_VEL
LIN {X 0,Y 150.357,Z 296.568,A -85,B 0,C 180,E1 -23884.032,E2 -23884.032} C_VEL
LIN {X 0,Y 150.223,Z 296.585,A -85,B 0,C 180,E1 -23887.459,E2 -23887.459} C_VEL
LIN {X 0,Y 150.157,Z 296.59,A -85,B 0,C 180,E1 -23891.505,E2 -23891.505} C_VEL
LIN {X 0,Y 150.129,Z 296.595,A -85,B 0,C 180,E1 -23895.394,E2 -23895.394} C_VEL
LIN {X 0,Y 150.144,Z 296.594,A -85,B 0,C 180,E1 -23899.054,E2 -23899.054} C_VEL
LIN {X 0,Y 150.182,Z 296.586,A -85,B 0,C 180,E1 -23902.706,E2 -23902.706} C_VEL
LIN {X 0,Y 150.217,Z 296.586,A -85,B 0,C 180,E1 -23907.366,E2 -23907.366} C_VEL
LIN {X 0,Y 150.246,Z 296.58,A -85,B 0,C 180,E1 -23912.716,E2 -23912.716} C_VEL
LIN {X 0,Y 150.352,Z 296.563,A -85,B 0,C 180,E1 -23919.206,E2 -23919.206} C_VEL
LIN {X 0,Y 150.362,Z 296.568,A -85,B 0,C 180,E1 -23923.711,E2 -23923.711} C_VEL
LIN {X 0,Y 150.612,Z 296.534,A -85,B 0,C 180,E1 -23929.24,E2 -23929.24} C_VEL
LIN {X 0,Y 150.704,Z 296.525,A -85,B 0,C 180,E1 -23931.956,E2 -23931.956} C_VEL
LIN {X 0,Y 151.216,Z 296.461,A -85,B 0,C 180,E1 -23939.998,E2 -23939.998} C_VEL
LIN {X 0,Y 150.743,Z 296.52,A -85,B 0,C 180,E1 -23948.038,E2 -23948.038} C_VEL
LIN {X 0,Y 150.604,Z 296.534,A -85,B 0,C 180,E1 -23951.489,E2 -23951.489} C_VEL
LIN {X 0,Y 150.371,Z 296.566,A -85,B 0,C 180,E1 -23956.283,E2 -23956.283} C_VEL
LIN {X 0,Y 150.364,Z 296.561,A -85,B 0,C 180,E1 -23960.806,E2 -23960.806} C_VEL
LIN {X 0,Y 150.241,Z 296.582,A -85,B 0,C 180,E1 -23967.28,E2 -23967.28} C_VEL
LIN {X 0,Y 150.215,Z 296.585,A -85,B 0,C 180,E1 -23972.632,E2 -23972.632} C_VEL
LIN {X 0,Y 150.212,Z 296.582,A -85,B 0,C 180,E1 -23977.459,E2 -23977.459} C_VEL
LIN {X 0,Y 150.207,Z 296.587,A -85,B 0,C 180,E1 -23981.529,E2 -23981.529} C_VEL
LIN {X 0,Y 150.246,Z 296.578,A -85,B 0,C 180,E1 -23985.441,E2 -23985.441} C_VEL
LIN {X 0,Y 150.224,Z 296.583,A -85,B 0,C 180,E1 -23989.083,E2 -23989.083} C_VEL
LIN {X 0,Y 150.23,Z 296.581,A -85,B 0,C 180,E1 -23992.678,E2 -23992.678} C_VEL
LIN {X 0,Y 150.212,Z 296.585,A -85,B 0,C 180,E1 -23997.365,E2 -23997.365} C_VEL
LIN {X 0,Y 150.239,Z 296.577,A -85,B 0,C 180,E1 -24002.717,E2 -24002.717} C_VEL
LIN {X 0,Y 150.345,Z 296.569,A -85,B 0,C 180,E1 -24009.206,E2 -24009.206} C_VEL
LIN {X 0,Y 150.376,Z 296.564,A -85,B 0,C 180,E1 -24013.715,E2 -24013.715} C_VEL
LIN {X 0,Y 150.647,Z 296.529,A -85,B 0,C 180,E1 -24019.245,E2 -24019.245} C_VEL
LIN {X 0,Y 150.733,Z 296.52,A -85,B 0,C 180,E1 -24021.959,E2 -24021.959} C_VEL
LIN {X 0,Y 151.211,Z 296.459,A -85,B 0,C 180,E1 -24029.999,E2 -24029.999} C_VEL
LIN {X 0,Y 150.737,Z 296.517,A -85,B 0,C 180,E1 -24038.04,E2 -24038.04} C_VEL
LIN {X 0,Y 150.605,Z 296.538,A -85,B 0,C 180,E1 -24041.502,E2 -24041.502} C_VEL
LIN {X 0,Y 150.362,Z 296.566,A -85,B 0,C 180,E1 -24048.743,E2 -24048.743} C_VEL
LIN {X 0,Y 150.369,Z 296.565,A -85,B 0,C 180,E1 -24048.919,E2 -24048.919} C_VEL
LIN {X 0,Y 158.994,Z 322.047,A -85,B 0,C 180,E1 -24051.496,E2 -24051.496} C_VEL
LIN {X 0,Y 156.934,Z 363.538,A -85,B 0,C 180,E1 -24053.843,E2 -24053.843} C_VEL
LIN {X 0,Y 156.078,Z 375.269,A -85,B 0,C 180,E1 -24054.97,E2 -24054.97} C_VEL
LIN {X 0,Y 154.928,Z 386.373,A -85,B 0,C 180,E1 -24056.59,E2 -24056.59} C_VEL
LIN {X 0,Y 153.828,Z 395.275,A -85,B 0,C 180,E1 -24058.293,E2 -24058.293} C_VEL
LIN {X 0,Y 152.693,Z 403.031,A -85,B 0,C 180,E1 -24060.14,E2 -24060.14} C_VEL
LIN {X 0,Y 151.278,Z 411.684,A -85,B 0,C 180,E1 -24062.686,E2 -24062.686} C_VEL
LIN {X 0,Y 149.97,Z 420.155,A -85,B 0,C 180,E1 -24065.857,E2 -24065.857} C_VEL
LIN {X 0,Y 148.927,Z 427.176,A -85,B 0,C 180,E1 -24069.267,E2 -24069.267} C_VEL
LIN {X 0,Y 148.253,Z 432.154,A -85,B 0,C 180,E1 -24072.264,E2 -24072.264} C_VEL
LIN {X 0,Y 147.785,Z 436.48,A -85,B 0,C 180,E1 -24075.505,E2 -24075.505} C_VEL
LIN {X 0,Y 147.682,Z 440.628,A -85,B 0,C 180,E1 -24079.587,E2 -24079.587} C_VEL
LIN {X 0,Y 148.19,Z 443.58,A -85,B 0,C 180,E1 -24083.727,E2 -24083.727} C_VEL
LIN {X 0,Y 149.397,Z 445.296,A -85,B 0,C 180,E1 -24087.859,E2 -24087.859} C_VEL
LIN {X 0,Y 151.448,Z 445.761,A -85,B 0,C 180,E1 -24092.354,E2 -24092.354} C_VEL
LIN {X 0,Y 153.813,Z 445.104,A -85,B 0,C 180,E1 -24096.037,E2 -24096.037} C_VEL
LIN {X 0,Y 157.072,Z 443.22,A -85,B 0,C 180,E1 -24099.983,E2 -24099.983} C_VEL
LIN {X 0,Y 161.049,Z 440.054,A -85,B 0,C 180,E1 -24103.744,E2 -24103.744} C_VEL
LIN {X 0,Y 165.688,Z 435.288,A -85,B 0,C 180,E1 -24107.307,E2 -24107.307} C_VEL
LIN {X 0,Y 169.623,Z 430.601,A -85,B 0,C 180,E1 -24109.86,E2 -24109.86} C_VEL
LIN {X 0,Y 173.07,Z 425.935,A -85,B 0,C 180,E1 -24111.895,E2 -24111.895} C_VEL
LIN {X 0,Y 177.275,Z 419.488,A -85,B 0,C 180,E1 -24114.082,E2 -24114.082} C_VEL
LIN {X 0,Y 181.049,Z 412.717,A -85,B 0,C 180,E1 -24115.92,E2 -24115.92} C_VEL
LIN {X 0,Y 184.539,Z 405.562,A -85,B 0,C 180,E1 -24117.452,E2 -24117.452} C_VEL
LIN {X 0,Y 187.924,Z 397.268,A -85,B 0,C 180,E1 -24118.885,E2 -24118.885} C_VEL
LIN {X 0,Y 191.271,Z 387.393,A -85,B 0,C 180,E1 -24120.178,E2 -24120.178} C_VEL
LIN {X 0,Y 193.973,Z 376.204,A -85,B 0,C 180,E1 -24121.27,E2 -24121.27} C_VEL
LIN {X 0,Y 195.701,Z 366.352,A -85,B 0,C 180,E1 -24121.924,E2 -24121.924} C_VEL
LIN {X 0,Y 196.96,Z 355.436,A -85,B 0,C 180,E1 -24122.461,E2 -24122.461} C_VEL
LIN {X 0,Y 192.097,Z 345.681,A -85,B 0,C 180,E1 -24126.402,E2 -24126.402} C_VEL
LIN {X 0,Y 189.132,Z 341.11,A -85,B 0,C 180,E1 -24129.258,E2 -24129.258} C_VEL
LIN {X 0,Y 186.725,Z 337.167,A -85,B 0,C 180,E1 -24132.199,E2 -24132.199} C_VEL
LIN {X 0,Y 184.478,Z 334.239,A -85,B 0,C 180,E1 -24135.718,E2 -24135.718} C_VEL
LIN {X 0,Y 183.908,Z 332.702,A -85,B 0,C 180,E1 -24137.188,E2 -24137.188} C_VEL
LIN {X 0,Y 182.364,Z 331.79,A -85,B 0,C 180,E1 -24142.669,E2 -24142.669} C_VEL
LIN {X 0,Y 182.687,Z 332.076,A -85,B 0,C 180,E1 -24147.495,E2 -24147.495} C_VEL
LIN {X 0,Y 184.381,Z 335.344,A -85,B 0,C 180,E1 -24152.517,E2 -24152.517} C_VEL
LIN {X 0,Y 187.316,Z 341.538,A -85,B 0,C 180,E1 -24157.28,E2 -24157.28} C_VEL
LIN {X 0,Y 189.786,Z 347.023,A -85,B 0,C 180,E1 -24160.159,E2 -24160.159} C_VEL
LIN {X 0,Y 192.197,Z 352.663,A -85,B 0,C 180,E1 -24162.562,E2 -24162.562} C_VEL
LIN {X 0,Y 194.479,Z 358.782,A -85,B 0,C 180,E1 -24164.595,E2 -24164.595} C_VEL
LIN {X 0,Y 195.792,Z 363.095,A -85,B 0,C 180,E1 -24165.765,E2 -24165.765} C_VEL
LIN {X 0,Y 195.768,Z 369.608,A -85,B 0,C 180,E1 -24166.382,E2 -24166.382} C_VEL
LIN {X 0,Y 193.766,Z 382.722,A -85,B 0,C 180,E1 -24167.021,E2 -24167.021} C_VEL
LIN {X 0,Y 191.355,Z 392.832,A -85,B 0,C 180,E1 -24167.752,E2 -24167.752} C_VEL
LIN {X 0,Y 188.626,Z 401.596,A -85,B 0,C 180,E1 -24168.599,E2 -24168.599} C_VEL
LIN {X 0,Y 185.112,Z 410.909,A -85,B 0,C 180,E1 -24169.804,E2 -24169.804} C_VEL
LIN {X 0,Y 179.919,Z 421.814,A -85,B 0,C 180,E1 -24171.678,E2 -24171.678} C_VEL
LIN {X 0,Y 176.236,Z 428.578,A -85,B 0,C 180,E1 -24173.262,E2 -24173.262} C_VEL
LIN {X 0,Y 172.264,Z 435.053,A -85,B 0,C 180,E1 -24175.17,E2 -24175.17} C_VEL
LIN {X 0,Y 167.625,Z 441.714,A -85,B 0,C 180,E1 -24177.687,E2 -24177.687} C_VEL
LIN {X 0,Y 163.398,Z 447.129,A -85,B 0,C 180,E1 -24180.356,E2 -24180.356} C_VEL
LIN {X 0,Y 160.29,Z 450.678,A -85,B 0,C 180,E1 -24182.59,E2 -24182.59} C_VEL
LIN {X 0,Y 156.235,Z 454.843,A -85,B 0,C 180,E1 -24186.119,E2 -24186.119} C_VEL
LIN {X 0,Y 153.978,Z 456.928,A -85,B 0,C 180,E1 -24188.585,E2 -24188.585} C_VEL
LIN {X 0,Y 152.027,Z 458.546,A -85,B 0,C 180,E1 -24191.12,E2 -24191.12} C_VEL
LIN {X 0,Y 150.567,Z 459.658,A -85,B 0,C 180,E1 -24193.737,E2 -24193.737} C_VEL
LIN {X 0,Y 149.4,Z 460.218,A -85,B 0,C 180,E1 -24196.397,E2 -24196.397} C_VEL
LIN {X 0,Y 148.612,Z 460.352,A -85,B 0,C 180,E1 -24199.097,E2 -24199.097} C_VEL
LIN {X 0,Y 148.149,Z 460.066,A -85,B 0,C 180,E1 -24201.819,E2 -24201.819} C_VEL
LIN {X 0,Y 148.068,Z 458.906,A -85,B 0,C 180,E1 -24205.408,E2 -24205.408} C_VEL
LIN {X 0,Y 148.151,Z 457.916,A -85,B 0,C 180,E1 -24207.282,E2 -24207.282} C_VEL
LIN {X 0,Y 148.267,Z 455.459,A -85,B 0,C 180,E1 -24210.706,E2 -24210.706} C_VEL
LIN {X 0,Y 147.943,Z 454.144,A -85,B 0,C 180,E1 -24212.136,E2 -24212.136} C_VEL
LIN {X 0,Y 146.619,Z 451.788,A -85,B 0,C 180,E1 -24214.192,E2 -24214.192} C_VEL
LIN {X 0,Y 144.82,Z 449.071,A -85,B 0,C 180,E1 -24216.163,E2 -24216.163} C_VEL
LIN {X 0,Y 142.239,Z 443.762,A -85,B 0,C 180,E1 -24219.409,E2 -24219.409} C_VEL
LIN {X 0,Y 141.906,Z 440.163,A -85,B 0,C 180,E1 -24221.336,E2 -24221.336} C_VEL
LIN {X 0,Y 142.653,Z 433.965,A -85,B 0,C 180,E1 -24224.261,E2 -24224.261} C_VEL
LIN {X 0,Y 143.78,Z 426.645,A -85,B 0,C 180,E1 -24227.055,E2 -24227.055} C_VEL
LIN {X 0,Y 145.064,Z 418.84,A -85,B 0,C 180,E1 -24229.456,E2 -24229.456} C_VEL
LIN {X 0,Y 146.204,Z 410.589,A -85,B 0,C 180,E1 -24231.502,E2 -24231.502} C_VEL
LIN {X 0,Y 147.931,Z 399.343,A -85,B 0,C 180,E1 -24233.632,E2 -24233.632} C_VEL
LIN {X 0,Y 149.124,Z 388.205,A -85,B 0,C 180,E1 -24235.098,E2 -24235.098} C_VEL
LIN {X 0,Y 149.933,Z 378.367,A -85,B 0,C 180,E1 -24235.986,E2 -24235.986} C_VEL
LIN {X 0,Y 150.737,Z 356.618,A -85,B 0,C 180,E1 -24237.323,E2 -24237.323} C_VEL
LIN {X 0,Y 147.545,Z 313.398,A -85,B 0,C 180,E1 -24240.407,E2 -24240.407} C_VEL
LIN {X 0,Y 144.047,Z 301.095,A -85,B 0,C 180,E1 -24241.675,E2 -24241.675} C_VEL
LIN {X 0,Y 143.317,Z 297.444,A -85,B 0,C 180,E1 -24244.201,E2 -24244.201} C_VEL
LIN {X 0,Y 143.081,Z 297.475,A -85,B 0,C 180,E1 -24249.684,E2 -24249.684} C_VEL
LIN {X 0,Y 143.06,Z 297.472,A -85,B 0,C 180,E1 -24253.453,E2 -24253.453} C_VEL
LIN {X 0,Y 143.042,Z 297.481,A -85,B 0,C 180,E1 -24257.475,E2 -24257.475} C_VEL
LIN {X 0,Y 143.078,Z 297.47,A -85,B 0,C 180,E1 -24261.806,E2 -24261.806} C_VEL
LIN {X 0,Y 143.184,Z 297.462,A -85,B 0,C 180,E1 -24267.319,E2 -24267.319} C_VEL
LIN {X 0,Y 143.192,Z 297.46,A -85,B 0,C 180,E1 -24272.061,E2 -24272.061} C_VEL
LIN {X 0,Y 143.278,Z 297.443,A -85,B 0,C 180,E1 -24278.744,E2 -24278.744} C_VEL
LIN {X 0,Y 143.302,Z 297.446,A -85,B 0,C 180,E1 -24282.885,E2 -24282.885} C_VEL
LIN {X 0,Y 143.538,Z 297.414,A -85,B 0,C 180,E1 -24288.703,E2 -24288.703} C_VEL
LIN {X 0,Y 143.626,Z 297.408,A -85,B 0,C 180,E1 -24291.556,E2 -24291.556} C_VEL
LIN {X 0,Y 144.175,Z 297.338,A -85,B 0,C 180,E1 -24299.998,E2 -24299.998} C_VEL
LIN {X 0,Y 143.662,Z 297.401,A -85,B 0,C 180,E1 -24308.437,E2 -24308.437} C_VEL
LIN {X 0,Y 143.546,Z 297.411,A -85,B 0,C 180,E1 -24311.71,E2 -24311.71} C_VEL
LIN {X 0,Y 143.312,Z 297.445,A -85,B 0,C 180,E1 -24317.109,E2 -24317.109} C_VEL
LIN {X 0,Y 143.29,Z 297.442,A -85,B 0,C 180,E1 -24321.269,E2 -24321.269} C_VEL
LIN {X 0,Y 143.187,Z 297.457,A -85,B 0,C 180,E1 -24327.935,E2 -24327.935} C_VEL
LIN {X 0,Y 143.165,Z 297.464,A -85,B 0,C 180,E1 -24333.433,E2 -24333.433} C_VEL
LIN {X 0,Y 143.102,Z 297.47,A -85,B 0,C 180,E1 -24339.673,E2 -24339.673} C_VEL
LIN {X 0,Y 143.151,Z 297.466,A -85,B 0,C 180,E1 -24343.415,E2 -24343.415} C_VEL
LIN {X 0,Y 143.152,Z 297.461,A -85,B 0,C 180,E1 -24347.423,E2 -24347.423} C_VEL
LIN {X 0,Y 143.134,Z 297.468,A -85,B 0,C 180,E1 -24351.773,E2 -24351.773} C_VEL
LIN {X 0,Y 143.18,Z 297.46,A -85,B 0,C 180,E1 -24357.321,E2 -24357.321} C_VEL
LIN {X 0,Y 143.185,Z 297.457,A -85,B 0,C 180,E1 -24362.061,E2 -24362.061} C_VEL
LIN {X 0,Y 143.271,Z 297.449,A -85,B 0,C 180,E1 -24368.744,E2 -24368.744} C_VEL
LIN {X 0,Y 143.31,Z 297.441,A -85,B 0,C 180,E1 -24372.888,E2 -24372.888} C_VEL
LIN {X 0,Y 143.588,Z 297.408,A -85,B 0,C 180,E1 -24378.709,E2 -24378.709} C_VEL
LIN {X 0,Y 143.654,Z 297.399,A -85,B 0,C 180,E1 -24381.56,E2 -24381.56} C_VEL
LIN {X 0,Y 144.17,Z 297.336,A -85,B 0,C 180,E1 -24389.999,E2 -24389.999} C_VEL
LIN {X 0,Y 143.658,Z 297.4,A -85,B 0,C 180,E1 -24398.439,E2 -24398.439} C_VEL
LIN {X 0,Y 143.541,Z 297.418,A -85,B 0,C 180,E1 -24401.712,E2 -24401.712} C_VEL
LIN {X 0,Y 143.343,Z 297.441,A -85,B 0,C 180,E1 -24408.12,E2 -24408.12} C_VEL
LIN {X 0,Y 152.059,Z 322.883,A -85,B 0,C 180,E1 -24410.813,E2 -24410.813} C_VEL
LIN {X 0,Y 150.014,Z 363.777,A -85,B 0,C 180,E1 -24413.237,E2 -24413.237} C_VEL
LIN {X 0,Y 149.203,Z 374.911,A -85,B 0,C 180,E1 -24414.339,E2 -24414.339} C_VEL
LIN {X 0,Y 147.963,Z 386.444,A -85,B 0,C 180,E1 -24416.073,E2 -24416.073} C_VEL
LIN {X 0,Y 146.818,Z 395.53,A -85,B 0,C 180,E1 -24417.888,E2 -24417.888} C_VEL
LIN {X 0,Y 145.687,Z 402.996,A -85,B 0,C 180,E1 -24419.741,E2 -24419.741} C_VEL
LIN {X 0,Y 144.386,Z 410.625,A -85,B 0,C 180,E1 -24422.053,E2 -24422.053} C_VEL
LIN {X 0,Y 143.212,Z 418.141,A -85,B 0,C 180,E1 -24424.86,E2 -24424.86} C_VEL
LIN {X 0,Y 141.916,Z 426.551,A -85,B 0,C 180,E1 -24428.861,E2 -24428.861} C_VEL
LIN {X 0,Y 141.259,Z 431.342,A -85,B 0,C 180,E1 -24431.734,E2 -24431.734} C_VEL
LIN {X 0,Y 140.673,Z 436.455,A -85,B 0,C 180,E1 -24435.622,E2 -24435.622} C_VEL
LIN {X 0,Y 140.597,Z 440.34,A -85,B 0,C 180,E1 -24439.475,E2 -24439.475} C_VEL
LIN {X 0,Y 141.008,Z 443.154,A -85,B 0,C 180,E1 -24443.27,E2 -24443.27} C_VEL
LIN {X 0,Y 142.033,Z 445.117,A -85,B 0,C 180,E1 -24447.262,E2 -24447.262} C_VEL
LIN {X 0,Y 143.802,Z 446.168,A -85,B 0,C 180,E1 -24451.603,E2 -24451.603} C_VEL
LIN {X 0,Y 146.354,Z 446.042,A -85,B 0,C 180,E1 -24455.833,E2 -24455.833} C_VEL
LIN {X 0,Y 150.489,Z 444.067,A -85,B 0,C 180,E1 -24460.921,E2 -24460.921} C_VEL
LIN {X 0,Y 153.847,Z 441.74,A -85,B 0,C 180,E1 -24464.095,E2 -24464.095} C_VEL
LIN {X 0,Y 157.59,Z 438.541,A -85,B 0,C 180,E1 -24467.118,E2 -24467.118} C_VEL
LIN {X 0,Y 161.909,Z 434.263,A -85,B 0,C 180,E1 -24470.003,E2 -24470.003} C_VEL
LIN {X 0,Y 167.362,Z 427.836,A -85,B 0,C 180,E1 -24473.191,E2 -24473.191} C_VEL
LIN {X 0,Y 172.736,Z 420.075,A -85,B 0,C 180,E1 -24475.903,E2 -24475.903} C_VEL
LIN {X 0,Y 176.662,Z 413.405,A -85,B 0,C 180,E1 -24477.722,E2 -24477.722} C_VEL
LIN {X 0,Y 180.839,Z 405.282,A -85,B 0,C 180,E1 -24479.445,E2 -24479.445} C_VEL
LIN {X 0,Y 185.098,Z 395.276,A -85,B 0,C 180,E1 -24481.09,E2 -24481.09} C_VEL
LIN {X 0,Y 188.405,Z 384.948,A -85,B 0,C 180,E1 -24482.346,E2 -24482.346} C_VEL
LIN {X 0,Y 190.726,Z 375.45,A -85,B 0,C 180,E1 -24483.2,E2 -24483.2} C_VEL
LIN {X 0,Y 192.448,Z 365.606,A -85,B 0,C 180,E1 -24483.825,E2 -24483.825} C_VEL
LIN {X 0,Y 193.202,Z 359.162,A -85,B 0,C 180,E1 -24484.174,E2 -24484.174} C_VEL
LIN {X 0,Y 189.602,Z 351.358,A -85,B 0,C 180,E1 -24487.468,E2 -24487.468} C_VEL
LIN {X 0,Y 187.045,Z 347.373,A -85,B 0,C 180,E1 -24490.089,E2 -24490.089} C_VEL
LIN {X 0,Y 184.867,Z 343.663,A -85,B 0,C 180,E1 -24493.026,E2 -24493.026} C_VEL
LIN {X 0,Y 182.956,Z 340.817,A -85,B 0,C 180,E1 -24496.408,E2 -24496.408} C_VEL
LIN {X 0,Y 182.588,Z 339.708,A -85,B 0,C 180,E1 -24497.449,E2 -24497.449} C_VEL
LIN {X 0,Y 181.174,Z 338.79,A -85,B 0,C 180,E1 -24502.827,E2 -24502.827} C_VEL
LIN {X 0,Y 181.459,Z 339.027,A -85,B 0,C 180,E1 -24507.212,E2 -24507.212} C_VEL
LIN {X 0,Y 182.932,Z 342.198,A -85,B 0,C 180,E1 -24512.034,E2 -24512.034} C_VEL
LIN {X 0,Y 185.453,Z 347.957,A -85,B 0,C 180,E1 -24516.508,E2 -24516.508} C_VEL
LIN {X 0,Y 187.52,Z 352.958,A -85,B 0,C 180,E1 -24519.197,E2 -24519.197} C_VEL
LIN {X 0,Y 189.958,Z 359.202,A -85,B 0,C 180,E1 -24521.887,E2 -24521.887} C_VEL
LIN {X 0,Y 192.303,Z 366.361,A -85,B 0,C 180,E1 -24524.149,E2 -24524.149} C_VEL
LIN {X 0,Y 192.269,Z 370.547,A -85,B 0,C 180,E1 -24524.578,E2 -24524.578} C_VEL
LIN {X 0,Y 190.195,Z 382.857,A -85,B 0,C 180,E1 -24525.198,E2 -24525.198} C_VEL
LIN {X 0,Y 187.77,Z 392.461,A -85,B 0,C 180,E1 -24525.886,E2 -24525.886} C_VEL
LIN {X 0,Y 184.71,Z 401.748,A -85,B 0,C 180,E1 -24526.776,E2 -24526.776} C_VEL
LIN {X 0,Y 180.442,Z 412.301,A -85,B 0,C 180,E1 -24528.166,E2 -24528.166} C_VEL
LIN {X 0,Y 175.637,Z 421.668,A -85,B 0,C 180,E1 -24529.819,E2 -24529.819} C_VEL
LIN {X 0,Y 171.768,Z 428.394,A -85,B 0,C 180,E1 -24531.395,E2 -24531.395} C_VEL
LIN {X 0,Y 167.562,Z 434.839,A -85,B 0,C 180,E1 -24533.297,E2 -24533.297} C_VEL
LIN {X 0,Y 163.608,Z 440.262,A -85,B 0,C 180,E1 -24535.309,E2 -24535.309} C_VEL
LIN {X 0,Y 159.001,Z 445.824,A -85,B 0,C 180,E1 -24537.968,E2 -24537.968} C_VEL
LIN {X 0,Y 154.042,Z 451.083,A -85,B 0,C 180,E1 -24541.378,E2 -24541.378} C_VEL
LIN {X 0,Y 149.779,Z 455.057,A -85,B 0,C 180,E1 -24545.021,E2 -24545.021} C_VEL
LIN {X 0,Y 147.405,Z 456.957,A -85,B 0,C 180,E1 -24547.579,E2 -24547.579} C_VEL
LIN {X 0,Y 145.312,Z 458.398,A -85,B 0,C 180,E1 -24550.212,E2 -24550.212} C_VEL
LIN {X 0,Y 143.734,Z 459.411,A -85,B 0,C 180,E1 -24552.941,E2 -24552.941} C_VEL
LIN {X 0,Y 142.496,Z 459.896,A -85,B 0,C 180,E1 -24555.724,E2 -24555.724} C_VEL
LIN {X 0,Y 141.632,Z 459.869,A -85,B 0,C 180,E1 -24558.553,E2 -24558.553} C_VEL
LIN {X 0,Y 141.147,Z 459.424,A -85,B 0,C 180,E1 -24561.41,E2 -24561.41} C_VEL
LIN {X 0,Y 141.035,Z 458.035,A -85,B 0,C 180,E1 -24565.317,E2 -24565.317} C_VEL
LIN {X 0,Y 141.129,Z 456.139,A -85,B 0,C 180,E1 -24568.574,E2 -24568.574} C_VEL
LIN {X 0,Y 141.246,Z 453.882,A -85,B 0,C 180,E1 -24571.426,E2 -24571.426} C_VEL
LIN {X 0,Y 141.288,Z 450.634,A -85,B 0,C 180,E1 -24574.516,E2 -24574.516} C_VEL
LIN {X 0,Y 141.469,Z 444.96,A -85,B 0,C 180,E1 -24578.572,E2 -24578.572} C_VEL
LIN {X 0,Y 141.906,Z 440.163,A -85,B 0,C 180,E1 -24581.336,E2 -24581.336} C_VEL
LIN {X 0,Y 141.7,Z 436.489,A -85,B 0,C 180,E1 -24583.146,E2 -24583.146} C_VEL
LIN {X 0,Y 139.844,Z 429.737,A -85,B 0,C 180,E1 -24585.959,E2 -24585.959} C_VEL
LIN {X 0,Y 138.124,Z 422.208,A -85,B 0,C 180,E1 -24588.617,E2 -24588.617} C_VEL
LIN {X 0,Y 138.18,Z 417.307,A -85,B 0,C 180,E1 -24590.079,E2 -24590.079} C_VEL
LIN {X 0,Y 139.659,Z 407.315,A -85,B 0,C 180,E1 -24592.564,E2 -24592.564} C_VEL
LIN {X 0,Y 141.212,Z 396.951,A -85,B 0,C 180,E1 -24594.438,E2 -24594.438} C_VEL
LIN {X 0,Y 142.227,Z 387.462,A -85,B 0,C 180,E1 -24595.716,E2 -24595.716} C_VEL
LIN {X 0,Y 143.046,Z 377.647,A -85,B 0,C 180,E1 -24596.636,E2 -24596.636} C_VEL
LIN {X 0,Y 143.876,Z 357.396,A -85,B 0,C 180,E1 -24597.941,E2 -24597.941} C_VEL
LIN {X 0,Y 140.833,Z 315.054,A -85,B 0,C 180,E1 -24601.091,E2 -24601.091} C_VEL
LIN {X 0,Y 136.755,Z 300.677,A -85,B 0,C 180,E1 -24602.694,E2 -24602.694} C_VEL
LIN {X 0,Y 136.245,Z 298.325,A -85,B 0,C 180,E1 -24604.463,E2 -24604.463} C_VEL
LIN {X 0,Y 136.058,Z 298.35,A -85,B 0,C 180,E1 -24609.208,E2 -24609.208} C_VEL
LIN {X 0,Y 136.001,Z 298.351,A -85,B 0,C 180,E1 -24613.656,E2 -24613.656} C_VEL
LIN {X 0,Y 135.987,Z 298.358,A -85,B 0,C 180,E1 -24617.786,E2 -24617.786} C_VEL
LIN {X 0,Y 136.027,Z 298.348,A -85,B 0,C 180,E1 -24621.681,E2 -24621.681} C_VEL
LIN {X 0,Y 136.058,Z 298.35,A -85,B 0,C 180,E1 -24625.738,E2 -24625.738} C_VEL
LIN {X 0,Y 136.148,Z 298.337,A -85,B 0,C 180,E1 -24632.314,E2 -24632.314} C_VEL
LIN {X 0,Y 136.245,Z 298.319,A -85,B 0,C 180,E1 -24638.831,E2 -24638.831} C_VEL
LIN {X 0,Y 136.269,Z 298.321,A -85,B 0,C 180,E1 -24645.054,E2 -24645.054} C_VEL
LIN {X 0,Y 136.432,Z 298.3,A -85,B 0,C 180,E1 -24648.162,E2 -24648.162} C_VEL
LIN {X 0,Y 136.551,Z 298.288,A -85,B 0,C 180,E1 -24651.115,E2 -24651.115} C_VEL
LIN {X 0,Y 137.132,Z 298.216,A -85,B 0,C 180,E1 -24659.998,E2 -24659.998} C_VEL
LIN {X 0,Y 136.589,Z 298.283,A -85,B 0,C 180,E1 -24668.877,E2 -24668.877} C_VEL
LIN {X 0,Y 136.49,Z 298.29,A -85,B 0,C 180,E1 -24671.952,E2 -24671.952} C_VEL
LIN {X 0,Y 136.252,Z 298.324,A -85,B 0,C 180,E1 -24678.025,E2 -24678.025} C_VEL
LIN {X 0,Y 136.21,Z 298.326,A -85,B 0,C 180,E1 -24681.761,E2 -24681.761} C_VEL
LIN {X 0,Y 136.097,Z 298.339,A -85,B 0,C 180,E1 -24688.614,E2 -24688.614} C_VEL
LIN {X 0,Y 136.076,Z 298.346,A -85,B 0,C 180,E1 -24694.616,E2 -24694.616} C_VEL
LIN {X 0,Y 136.069,Z 298.344,A -85,B 0,C 180,E1 -24699.218,E2 -24699.218} C_VEL
LIN {X 0,Y 136.087,Z 298.345,A -85,B 0,C 180,E1 -24703.697,E2 -24703.697} C_VEL
LIN {X 0,Y 136.101,Z 298.341,A -85,B 0,C 180,E1 -24707.833,E2 -24707.833} C_VEL
LIN {X 0,Y 136.086,Z 298.346,A -85,B 0,C 180,E1 -24711.704,E2 -24711.704} C_VEL
LIN {X 0,Y 136.087,Z 298.341,A -85,B 0,C 180,E1 -24715.715,E2 -24715.715} C_VEL
LIN {X 0,Y 136.141,Z 298.333,A -85,B 0,C 180,E1 -24722.315,E2 -24722.315} C_VEL
LIN {X 0,Y 136.238,Z 298.326,A -85,B 0,C 180,E1 -24728.832,E2 -24728.832} C_VEL
LIN {X 0,Y 136.278,Z 298.321,A -85,B 0,C 180,E1 -24735.057,E2 -24735.057} C_VEL
LIN {X 0,Y 136.491,Z 298.293,A -85,B 0,C 180,E1 -24738.114,E2 -24738.114} C_VEL
LIN {X 0,Y 136.582,Z 298.279,A -85,B 0,C 180,E1 -24741.119,E2 -24741.119} C_VEL
LIN {X 0,Y 137.127,Z 298.213,A -85,B 0,C 180,E1 -24749.999,E2 -24749.999} C_VEL
LIN {X 0,Y 136.585,Z 298.28,A -85,B 0,C 180,E1 -24758.879,E2 -24758.879} C_VEL
LIN {X 0,Y 136.484,Z 298.297,A -85,B 0,C 180,E1 -24761.954,E2 -24761.954} C_VEL
LIN {X 0,Y 136.301,Z 298.319,A -85,B 0,C 180,E1 -24767.245,E2 -24767.245} C_VEL
LIN {X 0,Y 145.231,Z 324.396,A -85,B 0,C 180,E1 -24770.168,E2 -24770.168} C_VEL
LIN {X 0,Y 143.088,Z 364.407,A -85,B 0,C 180,E1 -24772.664,E2 -24772.664} C_VEL
LIN {X 0,Y 142.149,Z 375.946,A -85,B 0,C 180,E1 -24773.877,E2 -24773.877} C_VEL
LIN {X 0,Y 141.048,Z 386.168,A -85,B 0,C 180,E1 -24775.485,E2 -24775.485} C_VEL
LIN {X 0,Y 139.895,Z 394.953,A -85,B 0,C 180,E1 -24777.284,E2 -24777.284} C_VEL
LIN {X 0,Y 138.751,Z 402.419,A -85,B 0,C 180,E1 -24779.176,E2 -24779.176} C_VEL
LIN {X 0,Y 137.383,Z 410.275,A -85,B 0,C 180,E1 -24781.623,E2 -24781.623} C_VEL
LIN {X 0,Y 136.24,Z 417.462,A -85,B 0,C 180,E1 -24784.38,E2 -24784.38} C_VEL
LIN {X 0,Y 135.144,Z 424.305,A -85,B 0,C 180,E1 -24787.605,E2 -24787.605} C_VEL
LIN {X 0,Y 134.145,Z 431.294,A -85,B 0,C 180,E1 -24791.745,E2 -24791.745} C_VEL
LIN {X 0,Y 133.556,Z 436.54,A -85,B 0,C 180,E1 -24795.866,E2 -24795.866} C_VEL
LIN {X 0,Y 133.49,Z 439.879,A -85,B 0,C 180,E1 -24799.172,E2 -24799.172} C_VEL
LIN {X 0,Y 133.729,Z 442.18,A -85,B 0,C 180,E1 -24802.025,E2 -24802.025} C_VEL
LIN {X 0,Y 134.667,Z 444.857,A -85,B 0,C 180,E1 -24806.614,E2 -24806.614} C_VEL
LIN {X 0,Y 137.025,Z 446.527,A -85,B 0,C 180,E1 -24812.512,E2 -24812.512} C_VEL
LIN {X 0,Y 139.257,Z 446.584,A -85,B 0,C 180,E1 -24816.191,E2 -24816.191} C_VEL
LIN {X 0,Y 142.145,Z 445.769,A -85,B 0,C 180,E1 -24819.947,E2 -24819.947} C_VEL
LIN {X 0,Y 146.177,Z 443.735,A -85,B 0,C 180,E1 -24824.058,E2 -24824.058} C_VEL
LIN {X 0,Y 150.907,Z 440.298,A -85,B 0,C 180,E1 -24827.952,E2 -24827.952} C_VEL
LIN {X 0,Y 156.32,Z 435.415,A -85,B 0,C 180,E1 -24831.52,E2 -24831.52} C_VEL
LIN {X 0,Y 161.352,Z 429.981,A -85,B 0,C 180,E1 -24834.379,E2 -24834.379} C_VEL
LIN {X 0,Y 166.618,Z 423.389,A -85,B 0,C 180,E1 -24836.98,E2 -24836.98} C_VEL
LIN {X 0,Y 172.297,Z 414.634,A -85,B 0,C 180,E1 -24839.505,E2 -24839.505} C_VEL
LIN {X 0,Y 176.453,Z 407.09,A -85,B 0,C 180,E1 -24841.142,E2 -24841.142} C_VEL
LIN {X 0,Y 179.964,Z 399.515,A -85,B 0,C 180,E1 -24842.46,E2 -24842.46} C_VEL
LIN {X 0,Y 183.403,Z 390.573,A -85,B 0,C 180,E1 -24843.667,E2 -24843.667} C_VEL
LIN {X 0,Y 186.73,Z 379.207,A -85,B 0,C 180,E1 -24844.861,E2 -24844.861} C_VEL
LIN {X 0,Y 189.017,Z 367.652,A -85,B 0,C 180,E1 -24845.634,E2 -24845.634} C_VEL
LIN {X 0,Y 189.665,Z 362.97,A -85,B 0,C 180,E1 -24845.922,E2 -24845.922} C_VEL
LIN {X 0,Y 187.289,Z 357.295,A -85,B 0,C 180,E1 -24848.433,E2 -24848.433} C_VEL
LIN {X 0,Y 185.066,Z 353.657,A -85,B 0,C 180,E1 -24850.947,E2 -24850.947} C_VEL
LIN {X 0,Y 183.27,Z 350.393,A -85,B 0,C 180,E1 -24853.548,E2 -24853.548} C_VEL
LIN {X 0,Y 181.455,Z 347.364,A -85,B 0,C 180,E1 -24857.131,E2 -24857.131} C_VEL
LIN {X 0,Y 181.124,Z 346.549,A -85,B 0,C 180,E1 -24858.086,E2 -24858.086} C_VEL
LIN {X 0,Y 179.989,Z 345.765,A -85,B 0,C 180,E1 -24862.985,E2 -24862.985} C_VEL
LIN {X 0,Y 180.304,Z 346.169,A -85,B 0,C 180,E1 -24867.401,E2 -24867.401} C_VEL
LIN {X 0,Y 181.459,Z 348.871,A -85,B 0,C 180,E1 -24871.417,E2 -24871.417} C_VEL
LIN {X 0,Y 183.632,Z 354.334,A -85,B 0,C 180,E1 -24875.723,E2 -24875.723} C_VEL
LIN {X 0,Y 185.336,Z 359.013,A -85,B 0,C 180,E1 -24878.258,E2 -24878.258} C_VEL
LIN {X 0,Y 187.584,Z 365.105,A -85,B 0,C 180,E1 -24880.931,E2 -24880.931} C_VEL
LIN {X 0,Y 189.006,Z 370.11,A -85,B 0,C 180,E1 -24882.555,E2 -24882.555} C_VEL
LIN {X 0,Y 188.694,Z 373.111,A -85,B 0,C 180,E1 -24882.771,E2 -24882.771} C_VEL
LIN {X 0,Y 186.76,Z 383.497,A -85,B 0,C 180,E1 -24883.325,E2 -24883.325} C_VEL
LIN {X 0,Y 184.32,Z 392.571,A -85,B 0,C 180,E1 -24883.966,E2 -24883.966} C_VEL
LIN {X 0,Y 180.695,Z 403.016,A -85,B 0,C 180,E1 -24884.975,E2 -24884.975} C_VEL
LIN {X 0,Y 175.931,Z 413.699,A -85,B 0,C 180,E1 -24886.444,E2 -24886.444} C_VEL
LIN {X 0,Y 170.963,Z 422.665,A -85,B 0,C 180,E1 -24888.088,E2 -24888.088} C_VEL
LIN {X 0,Y 166.351,Z 429.965,A -85,B 0,C 180,E1 -24889.89,E2 -24889.89} C_VEL
LIN {X 0,Y 160.962,Z 437.466,A -85,B 0,C 180,E1 -24892.32,E2 -24892.32} C_VEL
LIN {X 0,Y 154.973,Z 444.568,A -85,B 0,C 180,E1 -24895.469,E2 -24895.469} C_VEL
LIN {X 0,Y 151.307,Z 448.411,A -85,B 0,C 180,E1 -24897.715,E2 -24897.715} C_VEL
LIN {X 0,Y 146.294,Z 452.88,A -85,B 0,C 180,E1 -24901.29,E2 -24901.29} C_VEL
LIN {X 0,Y 143.388,Z 455.237,A -85,B 0,C 180,E1 -24903.826,E2 -24903.826} C_VEL
LIN {X 0,Y 140.856,Z 456.99,A -85,B 0,C 180,E1 -24906.476,E2 -24906.476} C_VEL
LIN {X 0,Y 138.644,Z 458.254,A -85,B 0,C 180,E1 -24909.218,E2 -24909.218} C_VEL
LIN {X 0,Y 136.935,Z 459.091,A -85,B 0,C 180,E1 -24912.066,E2 -24912.066} C_VEL
LIN {X 0,Y 135.603,Z 459.511,A -85,B 0,C 180,E1 -24914.982,E2 -24914.982} C_VEL
LIN {X 0,Y 134.677,Z 459.379,A -85,B 0,C 180,E1 -24917.953,E2 -24917.953} C_VEL
LIN {X 0,Y 134.14,Z 458.771,A -85,B 0,C 180,E1 -24920.958,E2 -24920.958} C_VEL
LIN {X 0,Y 133.997,Z 457.149,A -85,B 0,C 180,E1 -24925.249,E2 -24925.249} C_VEL
LIN {X 0,Y 134.105,Z 455.173,A -85,B 0,C 180,E1 -24928.499,E2 -24928.499} C_VEL
LIN {X 0,Y 134.221,Z 452.738,A -85,B 0,C 180,E1 -24931.501,E2 -24931.501} C_VEL
LIN {X 0,Y 134.246,Z 449.556,A -85,B 0,C 180,E1 -24934.56,E2 -24934.56} C_VEL
LIN {X 0,Y 134.413,Z 444.579,A -85,B 0,C 180,E1 -24938.268,E2 -24938.268} C_VEL
LIN {X 0,Y 134.855,Z 439.461,A -85,B 0,C 180,E1 -24941.351,E2 -24941.351} C_VEL
LIN {X 0,Y 135.578,Z 433.598,A -85,B 0,C 180,E1 -24944.255,E2 -24944.255} C_VEL
LIN {X 0,Y 136.863,Z 425.28,A -85,B 0,C 180,E1 -24947.559,E2 -24947.559} C_VEL
LIN {X 0,Y 138.18,Z 417.307,A -85,B 0,C 180,E1 -24950.079,E2 -24950.079} C_VEL
LIN {X 0,Y 138.309,Z 412.402,A -85,B 0,C 180,E1 -24951.446,E2 -24951.446} C_VEL
LIN {X 0,Y 136.941,Z 403.926,A -85,B 0,C 180,E1 -24953.504,E2 -24953.504} C_VEL
LIN {X 0,Y 135.351,Z 394.994,A -85,B 0,C 180,E1 -24955.232,E2 -24955.232} C_VEL
LIN {X 0,Y 135.131,Z 389.365,A -85,B 0,C 180,E1 -24956.044,E2 -24956.044} C_VEL
LIN {X 0,Y 136.04,Z 378.472,A -85,B 0,C 180,E1 -24957.186,E2 -24957.186} C_VEL
LIN {X 0,Y 136.958,Z 357.666,A -85,B 0,C 180,E1 -24958.611,E2 -24958.611} C_VEL
LIN {X 0,Y 133.996,Z 316.167,A -85,B 0,C 180,E1 -24961.891,E2 -24961.891} C_VEL
LIN {X 0,Y 129.429,Z 300.258,A -85,B 0,C 180,E1 -24963.787,E2 -24963.787} C_VEL
LIN {X 0,Y 129.154,Z 299.209,A -85,B 0,C 180,E1 -24964.793,E2 -24964.793} C_VEL
LIN {X 0,Y 128.956,Z 299.232,A -85,B 0,C 180,E1 -24970.843,E2 -24970.843} C_VEL
LIN {X 0,Y 128.919,Z 299.236,A -85,B 0,C 180,E1 -24975.128,E2 -24975.128} C_VEL
LIN {X 0,Y 128.938,Z 299.233,A -85,B 0,C 180,E1 -24979.737,E2 -24979.737} C_VEL
LIN {X 0,Y 128.961,Z 299.232,A -85,B 0,C 180,E1 -24984.831,E2 -24984.831} C_VEL
LIN {X 0,Y 129.019,Z 299.22,A -85,B 0,C 180,E1 -24990.64,E2 -24990.64} C_VEL
LIN {X 0,Y 129.032,Z 299.224,A -85,B 0,C 180,E1 -24994.165,E2 -24994.165} C_VEL
LIN {X 0,Y 129.109,Z 299.209,A -85,B 0,C 180,E1 -24997.726,E2 -24997.726} C_VEL
LIN {X 0,Y 129.154,Z 299.207,A -85,B 0,C 180,E1 -25000.941,E2 -25000.941} C_VEL
LIN {X 0,Y 129.377,Z 299.177,A -85,B 0,C 180,E1 -25007.901,E2 -25007.901} C_VEL
LIN {X 0,Y 129.475,Z 299.169,A -85,B 0,C 180,E1 -25010.625,E2 -25010.625} C_VEL
LIN {X 0,Y 130.087,Z 299.093,A -85,B 0,C 180,E1 -25019.997,E2 -25019.997} C_VEL
LIN {X 0,Y 129.515,Z 299.165,A -85,B 0,C 180,E1 -25029.366,E2 -25029.366} C_VEL
LIN {X 0,Y 129.392,Z 299.173,A -85,B 0,C 180,E1 -25032.545,E2 -25032.545} C_VEL
LIN {X 0,Y 129.165,Z 299.206,A -85,B 0,C 180,E1 -25039.051,E2 -25039.051} C_VEL
LIN {X 0,Y 129.109,Z 299.212,A -85,B 0,C 180,E1 -25042.395,E2 -25042.395} C_VEL
LIN {X 0,Y 129.033,Z 299.218,A -85,B 0,C 180,E1 -25049.371,E2 -25049.371} C_VEL
LIN {X 0,Y 128.992,Z 299.229,A -85,B 0,C 180,E1 -25055.189,E2 -25055.189} C_VEL
LIN {X 0,Y 129.002,Z 299.227,A -85,B 0,C 180,E1 -25060.822,E2 -25060.822} C_VEL
LIN {X 0,Y 129.02,Z 299.223,A -85,B 0,C 180,E1 -25065.079,E2 -25065.079} C_VEL
LIN {X 0,Y 129.009,Z 299.228,A -85,B 0,C 180,E1 -25069.696,E2 -25069.696} C_VEL
LIN {X 0,Y 129.019,Z 299.218,A -85,B 0,C 180,E1 -25074.789,E2 -25074.789} C_VEL
LIN {X 0,Y 129.046,Z 299.221,A -85,B 0,C 180,E1 -25080.649,E2 -25080.649} C_VEL
LIN {X 0,Y 129.102,Z 299.217,A -85,B 0,C 180,E1 -25087.726,E2 -25087.726} C_VEL
LIN {X 0,Y 129.154,Z 299.204,A -85,B 0,C 180,E1 -25090.943,E2 -25090.943} C_VEL
LIN {X 0,Y 129.41,Z 299.176,A -85,B 0,C 180,E1 -25097.819,E2 -25097.819} C_VEL
LIN {X 0,Y 129.508,Z 299.159,A -85,B 0,C 180,E1 -25100.63,E2 -25100.63} C_VEL
LIN {X 0,Y 130.082,Z 299.09,A -85,B 0,C 180,E1 -25109.999,E2 -25109.999} C_VEL
LIN {X 0,Y 129.51,Z 299.162,A -85,B 0,C 180,E1 -25119.368,E2 -25119.368} C_VEL
LIN {X 0,Y 129.388,Z 299.179,A -85,B 0,C 180,E1 -25122.548,E2 -25122.548} C_VEL
LIN {X 0,Y 129.254,Z 299.298,A -85,B 0,C 180,E1 -25126.321,E2 -25126.321} C_VEL
LIN {X 0,Y 138.283,Z 325.467,A -85,B 0,C 180,E1 -25129.429,E2 -25129.429} C_VEL
LIN {X 0,Y 136.182,Z 364.858,A -85,B 0,C 180,E1 -25132.018,E2 -25132.018} C_VEL
LIN {X 0,Y 135.047,Z 377.581,A -85,B 0,C 180,E1 -25133.47,E2 -25133.47} C_VEL
LIN {X 0,Y 133.963,Z 387.269,A -85,B 0,C 180,E1 -25135.11,E2 -25135.11} C_VEL
LIN {X 0,Y 132.809,Z 395.824,A -85,B 0,C 180,E1 -25136.977,E2 -25136.977} C_VEL
LIN {X 0,Y 131.477,Z 403.868,A -85,B 0,C 180,E1 -25139.164,E2 -25139.164} C_VEL
LIN {X 0,Y 129.915,Z 412.806,A -85,B 0,C 180,E1 -25142.212,E2 -25142.212} C_VEL
LIN {X 0,Y 128.527,Z 421.355,A -85,B 0,C 180,E1 -25145.958,E2 -25145.958} C_VEL
LIN {X 0,Y 127.533,Z 427.704,A -85,B 0,C 180,E1 -25149.516,E2 -25149.516} C_VEL
LIN {X 0,Y 126.681,Z 433.828,A -85,B 0,C 180,E1 -25153.85,E2 -25153.85} C_VEL
LIN {X 0,Y 126.385,Z 438.554,A -85,B 0,C 180,E1 -25158.145,E2 -25158.145} C_VEL
LIN {X 0,Y 126.667,Z 442.111,A -85,B 0,C 180,E1 -25162.391,E2 -25162.391} C_VEL
LIN {X 0,Y 127.515,Z 444.649,A -85,B 0,C 180,E1 -25166.557,E2 -25166.557} C_VEL
LIN {X 0,Y 128.951,Z 446.298,A -85,B 0,C 180,E1 -25170.69,E2 -25170.69} C_VEL
LIN {X 0,Y 131.408,Z 447.148,A -85,B 0,C 180,E1 -25175.391,E2 -25175.391} C_VEL
LIN {X 0,Y 134.668,Z 446.758,A -85,B 0,C 180,E1 -25179.942,E2 -25179.942} C_VEL
LIN {X 0,Y 138.734,Z 445.168,A -85,B 0,C 180,E1 -25184.253,E2 -25184.253} C_VEL
LIN {X 0,Y 144.089,Z 441.985,A -85,B 0,C 180,E1 -25188.752,E2 -25188.752} C_VEL
LIN {X 0,Y 150.174,Z 437.264,A -85,B 0,C 180,E1 -25192.728,E2 -25192.728} C_VEL
LIN {X 0,Y 155.597,Z 431.992,A -85,B 0,C 180,E1 -25195.753,E2 -25195.753} C_VEL
LIN {X 0,Y 160.697,Z 426.193,A -85,B 0,C 180,E1 -25198.215,E2 -25198.215} C_VEL
LIN {X 0,Y 164.769,Z 420.835,A -85,B 0,C 180,E1 -25200.002,E2 -25200.002} C_VEL
LIN {X 0,Y 169.41,Z 413.713,A -85,B 0,C 180,E1 -25201.903,E2 -25201.903} C_VEL
LIN {X 0,Y 174.541,Z 404.516,A -85,B 0,C 180,E1 -25203.755,E2 -25203.755} C_VEL
LIN {X 0,Y 178.793,Z 394.981,A -85,B 0,C 180,E1 -25205.21,E2 -25205.21} C_VEL
LIN {X 0,Y 181.887,Z 386.185,A -85,B 0,C 180,E1 -25206.234,E2 -25206.234} C_VEL
LIN {X 0,Y 184.498,Z 376.553,A -85,B 0,C 180,E1 -25207.078,E2 -25207.078} C_VEL
LIN {X 0,Y 186.363,Z 366.858,A -85,B 0,C 180,E1 -25207.698,E2 -25207.698} C_VEL
LIN {X 0,Y 184.995,Z 363.281,A -85,B 0,C 180,E1 -25209.445,E2 -25209.445} C_VEL
LIN {X 0,Y 183.107,Z 359.881,A -85,B 0,C 180,E1 -25211.866,E2 -25211.866} C_VEL
LIN {X 0,Y 181.622,Z 357.036,A -85,B 0,C 180,E1 -25214.182,E2 -25214.182} C_VEL
LIN {X 0,Y 179.957,Z 353.81,A -85,B 0,C 180,E1 -25217.96,E2 -25217.96} C_VEL
LIN {X 0,Y 179.342,Z 353.158,A -85,B 0,C 180,E1 -25219.868,E2 -25219.868} C_VEL
LIN {X 0,Y 178.849,Z 352.809,A -85,B 0,C 180,E1 -25225.341,E2 -25225.341} C_VEL
LIN {X 0,Y 179.174,Z 353.52,A -85,B 0,C 180,E1 -25227.834,E2 -25227.834} C_VEL
LIN {X 0,Y 180.04,Z 355.705,A -85,B 0,C 180,E1 -25230.915,E2 -25230.915} C_VEL
LIN {X 0,Y 181.858,Z 360.797,A -85,B 0,C 180,E1 -25234.959,E2 -25234.959} C_VEL
LIN {X 0,Y 183.272,Z 365.142,A -85,B 0,C 180,E1 -25237.338,E2 -25237.338} C_VEL
LIN {X 0,Y 185.156,Z 370.898,A -85,B 0,C 180,E1 -25239.88,E2 -25239.88} C_VEL
LIN {X 0,Y 185.731,Z 373.426,A -85,B 0,C 180,E1 -25240.761,E2 -25240.761} C_VEL
LIN {X 0,Y 183.862,Z 383.054,A -85,B 0,C 180,E1 -25241.298,E2 -25241.298} C_VEL
LIN {X 0,Y 181.22,Z 392.463,A -85,B 0,C 180,E1 -25241.956,E2 -25241.956} C_VEL
LIN {X 0,Y 177.508,Z 402.646,A -85,B 0,C 180,E1 -25242.921,E2 -25242.921} C_VEL
LIN {X 0,Y 172.242,Z 413.846,A -85,B 0,C 180,E1 -25244.437,E2 -25244.437} C_VEL
LIN {X 0,Y 167.737,Z 421.71,A -85,B 0,C 180,E1 -25245.85,E2 -25245.85} C_VEL
LIN {X 0,Y 163.445,Z 428.27,A -85,B 0,C 180,E1 -25247.374,E2 -25247.374} C_VEL
LIN {X 0,Y 158.78,Z 434.563,A -85,B 0,C 180,E1 -25249.243,E2 -25249.243} C_VEL
LIN {X 0,Y 153.308,Z 441.028,A -85,B 0,C 180,E1 -25251.768,E2 -25251.768} C_VEL
LIN {X 0,Y 149.217,Z 445.292,A -85,B 0,C 180,E1 -25253.934,E2 -25253.934} C_VEL
LIN {X 0,Y 145.381,Z 448.898,A -85,B 0,C 180,E1 -25256.227,E2 -25256.227} C_VEL
LIN {X 0,Y 140.112,Z 453.147,A -85,B 0,C 180,E1 -25259.896,E2 -25259.896} C_VEL
LIN {X 0,Y 137.069,Z 455.315,A -85,B 0,C 180,E1 -25262.52,E2 -25262.52} C_VEL
LIN {X 0,Y 134.369,Z 457.008,A -85,B 0,C 180,E1 -25265.266,E2 -25265.266} C_VEL
LIN {X 0,Y 132.025,Z 458.125,A -85,B 0,C 180,E1 -25268.124,E2 -25268.124} C_VEL
LIN {X 0,Y 130.173,Z 458.775,A -85,B 0,C 180,E1 -25271.1,E2 -25271.1} C_VEL
LIN {X 0,Y 128.74,Z 459.024,A -85,B 0,C 180,E1 -25274.161,E2 -25274.161} C_VEL
LIN {X 0,Y 127.746,Z 458.85,A -85,B 0,C 180,E1 -25277.288,E2 -25277.288} C_VEL
LIN {X 0,Y 127.13,Z 458.106,A -85,B 0,C 180,E1 -25280.455,E2 -25280.455} C_VEL
LIN {X 0,Y 126.972,Z 456.263,A -85,B 0,C 180,E1 -25285.102,E2 -25285.102} C_VEL
LIN {X 0,Y 127.176,Z 453.028,A -85,B 0,C 180,E1 -25290.001,E2 -25290.001} C_VEL
LIN {X 0,Y 127.172,Z 450.093,A -85,B 0,C 180,E1 -25293.169,E2 -25293.169} C_VEL
LIN {X 0,Y 127.336,Z 444.191,A -85,B 0,C 180,E1 -25297.932,E2 -25297.932} C_VEL
LIN {X 0,Y 127.766,Z 439.236,A -85,B 0,C 180,E1 -25301.101,E2 -25301.101} C_VEL
LIN {X 0,Y 128.481,Z 433.225,A -85,B 0,C 180,E1 -25304.25,E2 -25304.25} C_VEL
LIN {X 0,Y 129.773,Z 424.91,A -85,B 0,C 180,E1 -25307.736,E2 -25307.736} C_VEL
LIN {X 0,Y 131.193,Z 416.699,A -85,B 0,C 180,E1 -25310.464,E2 -25310.464} C_VEL
LIN {X 0,Y 132.958,Z 405.231,A -85,B 0,C 180,E1 -25313.356,E2 -25313.356} C_VEL
LIN {X 0,Y 134.395,Z 395.505,A -85,B 0,C 180,E1 -25315.144,E2 -25315.144} C_VEL
LIN {X 0,Y 135.131,Z 389.365,A -85,B 0,C 180,E1 -25316.044,E2 -25316.044} C_VEL
LIN {X 0,Y 135.006,Z 383.692,A -85,B 0,C 180,E1 -25316.773,E2 -25316.773} C_VEL
LIN {X 0,Y 133.93,Z 378.069,A -85,B 0,C 180,E1 -25317.444,E2 -25317.444} C_VEL
LIN {X 0,Y 131.033,Z 366.825,A -85,B 0,C 180,E1 -25318.622,E2 -25318.622} C_VEL
LIN {X 0,Y 130.181,Z 361.063,A -85,B 0,C 180,E1 -25319.117,E2 -25319.117} C_VEL
LIN {X 0,Y 130.113,Z 359.116,A -85,B 0,C 180,E1 -25319.265,E2 -25319.265} C_VEL
LIN {X 0,Y 127.356,Z 317.912,A -85,B 0,C 180,E1 -25322.693,E2 -25322.693} C_VEL
LIN {X 0,Y 122.113,Z 300.085,A -85,B 0,C 180,E1 -25324.91,E2 -25324.91} C_VEL
LIN {X 0,Y 121.889,Z 300.111,A -85,B 0,C 180,E1 -25331.443,E2 -25331.443} C_VEL
LIN {X 0,Y 121.867,Z 300.116,A -85,B 0,C 180,E1 -25338.564,E2 -25338.564} C_VEL
LIN {X 0,Y 121.913,Z 300.11,A -85,B 0,C 180,E1 -25344.794,E2 -25344.794} C_VEL
LIN {X 0,Y 121.929,Z 300.103,A -85,B 0,C 180,E1 -25349.837,E2 -25349.837} C_VEL
LIN {X 0,Y 121.985,Z 300.1,A -85,B 0,C 180,E1 -25356.213,E2 -25356.213} C_VEL
LIN {X 0,Y 122.047,Z 300.091,A -85,B 0,C 180,E1 -25359.784,E2 -25359.784} C_VEL
LIN {X 0,Y 122.24,Z 300.064,A -85,B 0,C 180,E1 -25366.702,E2 -25366.702} C_VEL
LIN {X 0,Y 122.407,Z 300.05,A -85,B 0,C 180,E1 -25370.079,E2 -25370.079} C_VEL
LIN {X 0,Y 122.597,Z 300.022,A -85,B 0,C 180,E1 -25376.711,E2 -25376.711} C_VEL
LIN {X 0,Y 123.041,Z 299.971,A -85,B 0,C 180,E1 -25379.997,E2 -25379.997} C_VEL
LIN {X 0,Y 122.415,Z 300.044,A -85,B 0,C 180,E1 -25387.173,E2 -25387.173} C_VEL
LIN {X 0,Y 122.362,Z 300.048,A -85,B 0,C 180,E1 -25392.47,E2 -25392.47} C_VEL
LIN {X 0,Y 122.055,Z 300.087,A -85,B 0,C 180,E1 -25400.208,E2 -25400.208} C_VEL
LIN {X 0,Y 121.984,Z 300.102,A -85,B 0,C 180,E1 -25403.781,E2 -25403.781} C_VEL
LIN {X 0,Y 121.939,Z 300.103,A -85,B 0,C 180,E1 -25410.171,E2 -25410.171} C_VEL
LIN {X 0,Y 121.915,Z 300.107,A -85,B 0,C 180,E1 -25416.191,E2 -25416.191} C_VEL
LIN {X 0,Y 121.932,Z 300.109,A -85,B 0,C 180,E1 -25421.47,E2 -25421.47} C_VEL
LIN {X 0,Y 121.937,Z 300.107,A -85,B 0,C 180,E1 -25428.522,E2 -25428.522} C_VEL
LIN {X 0,Y 121.971,Z 300.096,A -85,B 0,C 180,E1 -25434.816,E2 -25434.816} C_VEL
LIN {X 0,Y 121.937,Z 300.109,A -85,B 0,C 180,E1 -25439.824,E2 -25439.824} C_VEL
LIN {X 0,Y 121.978,Z 300.103,A -85,B 0,C 180,E1 -25446.214,E2 -25446.214} C_VEL
LIN {X 0,Y 122.043,Z 300.092,A -85,B 0,C 180,E1 -25449.786,E2 -25449.786} C_VEL
LIN {X 0,Y 122.258,Z 300.068,A -85,B 0,C 180,E1 -25456.706,E2 -25456.706} C_VEL
LIN {X 0,Y 122.438,Z 300.04,A -85,B 0,C 180,E1 -25460.084,E2 -25460.084} C_VEL
LIN {X 0,Y 122.598,Z 300.023,A -85,B 0,C 180,E1 -25466.713,E2 -25466.713} C_VEL
LIN {X 0,Y 123.036,Z 299.967,A -85,B 0,C 180,E1 -25469.999,E2 -25469.999} C_VEL
LIN {X 0,Y 122.439,Z 300.039,A -85,B 0,C 180,E1 -25476.591,E2 -25476.591} C_VEL
LIN {X 0,Y 122.44,Z 300.045,A -85,B 0,C 180,E1 -25479.915,E2 -25479.915} C_VEL
LIN {X 0,Y 122.221,Z 300.175,A -85,B 0,C 180,E1 -25485.294,E2 -25485.294} C_VEL
LIN {X 0,Y 131.368,Z 326.536,A -85,B 0,C 180,E1 -25488.621,E2 -25488.621} C_VEL
LIN {X 0,Y 129.273,Z 365.041,A -85,B 0,C 180,E1 -25491.299,E2 -25491.299} C_VEL
LIN {X 0,Y 128.323,Z 375.93,A -85,B 0,C 180,E1 -25492.542,E2 -25492.542} C_VEL
LIN {X 0,Y 126.995,Z 387.361,A -85,B 0,C 180,E1 -25494.521,E2 -25494.521} C_VEL
LIN {X 0,Y 125.753,Z 396.372,A -85,B 0,C 180,E1 -25496.601,E2 -25496.601} C_VEL
LIN {X 0,Y 124.151,Z 405.348,A -85,B 0,C 180,E1 -25499.223,E2 -25499.223} C_VEL
LIN {X 0,Y 122.571,Z 414.317,A -85,B 0,C 180,E1 -25502.544,E2 -25502.544} C_VEL
LIN {X 0,Y 121.131,Z 422.873,A -85,B 0,C 180,E1 -25506.704,E2 -25506.704} C_VEL
LIN {X 0,Y 120.238,Z 429.141,A -85,B 0,C 180,E1 -25510.553,E2 -25510.553} C_VEL
LIN {X 0,Y 119.594,Z 433.686,A -85,B 0,C 180,E1 -25513.963,E2 -25513.963} C_VEL
LIN {X 0,Y 119.308,Z 437.446,A -85,B 0,C 180,E1 -25517.362,E2 -25517.362} C_VEL
LIN {X 0,Y 119.514,Z 441.469,A -85,B 0,C 180,E1 -25522.022,E2 -25522.022} C_VEL
LIN {X 0,Y 120.025,Z 443.569,A -85,B 0,C 180,E1 -25525.058,E2 -25525.058} C_VEL
LIN {X 0,Y 121.517,Z 446.01,A -85,B 0,C 180,E1 -25530.169,E2 -25530.169} C_VEL
LIN {X 0,Y 122.625,Z 446.875,A -85,B 0,C 180,E1 -25532.713,E2 -25532.713} C_VEL
LIN {X 0,Y 124.942,Z 447.559,A -85,B 0,C 180,E1 -25536.815,E2 -25536.815} C_VEL
LIN {X 0,Y 127.829,Z 447.428,A -85,B 0,C 180,E1 -25540.742,E2 -25540.742} C_VEL
LIN {X 0,Y 131.288,Z 446.489,A -85,B 0,C 180,E1 -25544.478,E2 -25544.478} C_VEL
LIN {X 0,Y 136.149,Z 444.273,A -85,B 0,C 180,E1 -25548.738,E2 -25548.738} C_VEL
LIN {X 0,Y 141.725,Z 440.708,A -85,B 0,C 180,E1 -25552.634,E2 -25552.634} C_VEL
LIN {X 0,Y 146.53,Z 436.975,A -85,B 0,C 180,E1 -25555.443,E2 -25555.443} C_VEL
LIN {X 0,Y 151.312,Z 432.575,A -85,B 0,C 180,E1 -25557.933,E2 -25557.933} C_VEL
LIN {X 0,Y 155.875,Z 427.779,A -85,B 0,C 180,E1 -25560.002,E2 -25560.002} C_VEL
LIN {X 0,Y 160.367,Z 422.365,A -85,B 0,C 180,E1 -25561.887,E2 -25561.887} C_VEL
LIN {X 0,Y 164.918,Z 415.975,A -85,B 0,C 180,E1 -25563.667,E2 -25563.667} C_VEL
LIN {X 0,Y 169.365,Z 408.773,A -85,B 0,C 180,E1 -25565.204,E2 -25565.204} C_VEL
LIN {X 0,Y 173.886,Z 399.943,A -85,B 0,C 180,E1 -25566.684,E2 -25566.684} C_VEL
LIN {X 0,Y 177.682,Z 390.838,A -85,B 0,C 180,E1 -25567.843,E2 -25567.843} C_VEL
LIN {X 0,Y 181.141,Z 379.922,A -85,B 0,C 180,E1 -25568.93,E2 -25568.93} C_VEL
LIN {X 0,Y 183.205,Z 370.698,A -85,B 0,C 180,E1 -25569.579,E2 -25569.579} C_VEL
LIN {X 0,Y 181.468,Z 366.721,A -85,B 0,C 180,E1 -25572.245,E2 -25572.245} C_VEL
LIN {X 0,Y 180.048,Z 363.726,A -85,B 0,C 180,E1 -25574.791,E2 -25574.791} C_VEL
LIN {X 0,Y 178.402,Z 360.298,A -85,B 0,C 180,E1 -25579.016,E2 -25579.016} C_VEL
LIN {X 0,Y 177.607,Z 359.79,A -85,B 0,C 180,E1 -25584.482,E2 -25584.482} C_VEL
LIN {X 0,Y 177.911,Z 360.305,A -85,B 0,C 180,E1 -25587.289,E2 -25587.289} C_VEL
LIN {X 0,Y 178.587,Z 362.318,A -85,B 0,C 180,E1 -25590.224,E2 -25590.224} C_VEL
LIN {X 0,Y 180.1,Z 367.19,A -85,B 0,C 180,E1 -25594.143,E2 -25594.143} C_VEL
LIN {X 0,Y 181.189,Z 371.1,A -85,B 0,C 180,E1 -25596.313,E2 -25596.313} C_VEL
LIN {X 0,Y 182.562,Z 376.47,A -85,B 0,C 180,E1 -25598.774,E2 -25598.774} C_VEL
LIN {X 0,Y 182.452,Z 377.769,A -85,B 0,C 180,E1 -25598.933,E2 -25598.933} C_VEL
LIN {X 0,Y 179.709,Z 388.489,A -85,B 0,C 180,E1 -25599.568,E2 -25599.568} C_VEL
LIN {X 0,Y 176.334,Z 398.17,A -85,B 0,C 180,E1 -25600.354,E2 -25600.354} C_VEL
LIN {X 0,Y 172.889,Z 406.218,A -85,B 0,C 180,E1 -25601.236,E2 -25601.236} C_VEL
LIN {X 0,Y 168.12,Z 415.375,A -85,B 0,C 180,E1 -25602.544,E2 -25602.544} C_VEL
LIN {X 0,Y 163.452,Z 422.877,A -85,B 0,C 180,E1 -25603.931,E2 -25603.931} C_VEL
LIN {X 0,Y 157.164,Z 431.617,A -85,B 0,C 180,E1 -25606.124,E2 -25606.124} C_VEL
LIN {X 0,Y 151.231,Z 438.547,A -85,B 0,C 180,E1 -25608.532,E2 -25608.532} C_VEL
LIN {X 0,Y 145.707,Z 444.144,A -85,B 0,C 180,E1 -25611.17,E2 -25611.17} C_VEL
LIN {X 0,Y 141.479,Z 447.891,A -85,B 0,C 180,E1 -25613.41,E2 -25613.41} C_VEL
LIN {X 0,Y 135.789,Z 452.235,A -85,B 0,C 180,E1 -25617.083,E2 -25617.083} C_VEL
LIN {X 0,Y 130.815,Z 455.386,A -85,B 0,C 180,E1 -25621.086,E2 -25621.086} C_VEL
LIN {X 0,Y 127.954,Z 456.896,A -85,B 0,C 180,E1 -25623.935,E2 -25623.935} C_VEL
LIN {X 0,Y 125.464,Z 457.963,A -85,B 0,C 180,E1 -25626.915,E2 -25626.915} C_VEL
LIN {X 0,Y 123.455,Z 458.466,A -85,B 0,C 180,E1 -25630.029,E2 -25630.029} C_VEL
LIN {X 0,Y 120.84,Z 458.195,A -85,B 0,C 180,E1 -25636.549,E2 -25636.549} C_VEL
LIN {X 0,Y 120.135,Z 457.419,A -85,B 0,C 180,E1 -25639.893,E2 -25639.893} C_VEL
LIN {X 0,Y 119.96,Z 455.308,A -85,B 0,C 180,E1 -25644.875,E2 -25644.875} C_VEL
LIN {X 0,Y 120.092,Z 453.164,A -85,B 0,C 180,E1 -25648.324,E2 -25648.324} C_VEL
LIN {X 0,Y 120.186,Z 450.364,A -85,B 0,C 180,E1 -25651.676,E2 -25651.676} C_VEL
LIN {X 0,Y 120.232,Z 444.882,A -85,B 0,C 180,E1 -25656.714,E2 -25656.714} C_VEL
LIN {X 0,Y 120.694,Z 438.781,A -85,B 0,C 180,E1 -25660.909,E2 -25660.909} C_VEL
LIN {X 0,Y 121.393,Z 432.786,A -85,B 0,C 180,E1 -25664.245,E2 -25664.245} C_VEL
LIN {X 0,Y 122.708,Z 424.504,A -85,B 0,C 180,E1 -25667.93,E2 -25667.93} C_VEL
LIN {X 0,Y 124.102,Z 416.58,A -85,B 0,C 180,E1 -25670.729,E2 -25670.729} C_VEL
LIN {X 0,Y 125.668,Z 406.642,A -85,B 0,C 180,E1 -25673.483,E2 -25673.483} C_VEL
LIN {X 0,Y 127.314,Z 396.335,A -85,B 0,C 180,E1 -25675.548,E2 -25675.548} C_VEL
LIN {X 0,Y 128.377,Z 386.9,A -85,B 0,C 180,E1 -25676.959,E2 -25676.959} C_VEL
LIN {X 0,Y 129.219,Z 377.175,A -85,B 0,C 180,E1 -25677.976,E2 -25677.976} C_VEL
LIN {X 0,Y 130.113,Z 359.116,A -85,B 0,C 180,E1 -25679.265,E2 -25679.265} C_VEL
LIN {X 0,Y 129.329,Z 353.404,A -85,B 0,C 180,E1 -25679.779,E2 -25679.779} C_VEL
LIN {X 0,Y 125.899,Z 344.43,A -85,B 0,C 180,E1 -25680.871,E2 -25680.871} C_VEL
LIN {X 0,Y 122.291,Z 335.476,A -85,B 0,C 180,E1 -25682.031,E2 -25682.031} C_VEL
LIN {X 0,Y 121.253,Z 329.779,A -85,B 0,C 180,E1 -25682.624,E2 -25682.624} C_VEL
LIN {X 0,Y 120.677,Z 319.547,A -85,B 0,C 180,E1 -25683.53,E2 -25683.53} C_VEL
LIN {X 0,Y 116.1,Z 304.081,A -85,B 0,C 180,E1 -25685.564,E2 -25685.564} C_VEL
LIN {X 0,Y 114.971,Z 300.974,A -85,B 0,C 180,E1 -25686.143,E2 -25686.143} C_VEL
LIN {X 0,Y 114.797,Z 300.991,A -85,B 0,C 180,E1 -25692.718,E2 -25692.718} C_VEL
LIN {X 0,Y 114.791,Z 300.999,A -85,B 0,C 180,E1 -25697.661,E2 -25697.661} C_VEL
LIN {X 0,Y 114.788,Z 300.994,A -85,B 0,C 180,E1 -25702.744,E2 -25702.744} C_VEL
LIN {X 0,Y 114.859,Z 300.986,A -85,B 0,C 180,E1 -25708.941,E2 -25708.941} C_VEL
LIN {X 0,Y 114.95,Z 300.976,A -85,B 0,C 180,E1 -25716.504,E2 -25716.504} C_VEL
LIN {X 0,Y 115.012,Z 300.971,A -85,B 0,C 180,E1 -25722.207,E2 -25722.207} C_VEL
LIN {X 0,Y 115.256,Z 300.934,A -85,B 0,C 180,E1 -25727.325,E2 -25727.325} C_VEL
LIN {X 0,Y 115.365,Z 300.926,A -85,B 0,C 180,E1 -25732.999,E2 -25732.999} C_VEL
LIN {X 0,Y 115.992,Z 300.849,A -85,B 0,C 180,E1 -25739.997,E2 -25739.997} C_VEL
LIN {X 0,Y 115.382,Z 300.923,A -85,B 0,C 180,E1 -25747.064,E2 -25747.064} C_VEL
LIN {X 0,Y 115.283,Z 300.93,A -85,B 0,C 180,E1 -25752.734,E2 -25752.734} C_VEL
LIN {X 0,Y 115.018,Z 300.97,A -85,B 0,C 180,E1 -25757.786,E2 -25757.786} C_VEL
LIN {X 0,Y 114.947,Z 300.978,A -85,B 0,C 180,E1 -25763.492,E2 -25763.492} C_VEL
LIN {X 0,Y 114.866,Z 300.986,A -85,B 0,C 180,E1 -25771.065,E2 -25771.065} C_VEL
LIN {X 0,Y 114.818,Z 300.989,A -85,B 0,C 180,E1 -25777.737,E2 -25777.737} C_VEL
LIN {X 0,Y 114.857,Z 300.99,A -85,B 0,C 180,E1 -25782.754,E2 -25782.754} C_VEL
LIN {X 0,Y 114.865,Z 300.985,A -85,B 0,C 180,E1 -25787.698,E2 -25787.698} C_VEL
LIN {X 0,Y 114.85,Z 300.989,A -85,B 0,C 180,E1 -25792.697,E2 -25792.697} C_VEL
